   S711A_WELD_BUFF_DATA1.RBT13_BT_CODE_NO := W#16#0;
   S711A_WELD_BUFF_DATA1.RBT13_WELD_COUNT := W#16#0;
   S711A_WELD_BUFF_DATA1.RBT14_BT_CODE_NO := W#16#0;
   S711A_WELD_BUFF_DATA1.RBT14_WELD_COUNT := W#16#0;
   S711A_WELD_BUFF_DATA1.RBT15_BT_CODE_NO := W#16#0;
   S711A_WELD_BUFF_DATA1.RBT15_WELD_COUNT := W#16#0;
   S711A_WELD_BUFF_DATA1.RBT16_BT_CODE_NO := W#16#0;
   S711A_WELD_BUFF_DATA1.RBT16_WELD_COUNT := W#16#0;
   S711A_WELD_BUFF_DATA1.RBT17_BT_CODE_NO := W#16#0;
   S711A_WELD_BUFF_DATA1.RBT17_WELD_COUNT := W#16#0;
   S711A_WELD_BUFF_DATA1.RBT18_BT_CODE_NO := W#16#0;
   S711A_WELD_BUFF_DATA1.RBT18_WELD_COUNT := W#16#0;
   S711A_WELD_BUFF_DATA1.RBT19_BT_CODE_NO := W#16#0;
   S711A_WELD_BUFF_DATA1.RBT19_WELD_COUNT := W#16#0;
   S711A_WELD_BUFF_DATA1.RBT20_BT_CODE_NO := W#16#0;
   S711A_WELD_BUFF_DATA1.RBT20_WELD_COUNT := W#16#0;
   S711A_WELD_BUFF_DATA1.RBT21_BT_CODE_NO := W#16#0;
   S711A_WELD_BUFF_DATA1.RBT21_WELD_COUNT := W#16#0;
   S711A_WELD_BUFF_DATA1.RBT22_BT_CODE_NO := W#16#0;
   S711A_WELD_BUFF_DATA1.RBT22_WELD_COUNT := W#16#0;
   S711A_WELD_BUFF_DATA1.RBT23_BT_CODE_NO := W#16#0;
   S711A_WELD_BUFF_DATA1.RBT23_WELD_COUNT := W#16#0;
   S711A_WELD_BUFF_DATA1.RBT24_BT_CODE_NO := W#16#0;
   S711A_WELD_BUFF_DATA1.RBT24_WELD_COUNT := W#16#0;
   S711A_WELD_BUFF_DATA1.WELD_DETERMINES_RESULT := W#16#0;
   S711A_WELD_BUFF_DATA1.WELD_CHECK_SUM := W#16#0;
   S711A_WELD_BUFF_DATA1.SPARE1 := W#16#0;
   S711A_WELD_BUFF_DATA2.STATION_MAIN := W#16#0;
   S711A_WELD_BUFF_DATA2.DISTINCTION_LH_RH := W#16#0;
   S711A_WELD_BUFF_DATA2.STAION_NUMBER := W#16#0;
   S711A_WELD_BUFF_DATA2.VIN_NUMBER1 := W#16#0;
   S711A_WELD_BUFF_DATA2.VIN_NUMBER2 := W#16#0;
   S711A_WELD_BUFF_DATA2.VIN_NUMBER3 := W#16#0;
   S711A_WELD_BUFF_DATA2.VIN_NUMBER4 := W#16#0;
   S711A_WELD_BUFF_DATA2.SEQ_NUMBER1 := W#16#0;
   S711A_WELD_BUFF_DATA2.SEQ_NUMBER2 := W#16#0;
   S711A_WELD_BUFF_DATA2.RBT1_BT_CODE_NO := W#16#0;
   S711A_WELD_BUFF_DATA2.RBT1_WELD_COUNT := W#16#0;
   S711A_WELD_BUFF_DATA2.RBT2_BT_CODE_NO := W#16#0;
   S711A_WELD_BUFF_DATA2.RBT2_WELD_COUNT := W#16#0;
   S711A_WELD_BUFF_DATA2.RBT3_BT_CODE_NO := W#16#0;
   S711A_WELD_BUFF_DATA2.RBT3_WELD_COUNT := W#16#0;
   S711A_WELD_BUFF_DATA2.RBT4_BT_CODE_NO := W#16#0;
   S711A_WELD_BUFF_DATA2.RBT4_WELD_COUNT := W#16#0;
   S711A_WELD_BUFF_DATA2.RBT5_BT_CODE_NO := W#16#0;
   S711A_WELD_BUFF_DATA2.RBT5_WELD_COUNT := W#16#0;
   S711A_WELD_BUFF_DATA2.RBT6_BT_CODE_NO := W#16#0;
   S711A_WELD_BUFF_DATA2.RBT6_WELD_COUNT := W#16#0;
   S711A_WELD_BUFF_DATA2.RBT7_BT_CODE_NO := W#16#0;
   S711A_WELD_BUFF_DATA2.RBT7_WELD_COUNT := W#16#0;
   S711A_WELD_BUFF_DATA2.RBT8_BT_CODE_NO := W#16#0;
   S711A_WELD_BUFF_DATA2.RBT8_WELD_COUNT := W#16#0;
   S711A_WELD_BUFF_DATA2.RBT9_BT_CODE_NO := W#16#0;
   S711A_WELD_BUFF_DATA2.RBT9_WELD_COUNT := W#16#0;
   S711A_WELD_BUFF_DATA2.RBT10_BT_CODE_NO := W#16#0;
   S711A_WELD_BUFF_DATA2.RBT10_WELD_COUNT := W#16#0;
   S711A_WELD_BUFF_DATA2.RBT11_BT_CODE_NO := W#16#0;
   S711A_WELD_BUFF_DATA2.RBT11_WELD_COUNT := W#16#0;
   S711A_WELD_BUFF_DATA2.RBT12_BT_CODE_NO := W#16#0;
   S711A_WELD_BUFF_DATA2.RBT12_WELD_COUNT := W#16#0;
   S711A_WELD_BUFF_DATA2.RBT13_BT_CODE_NO := W#16#0;
   S711A_WELD_BUFF_DATA2.RBT13_WELD_COUNT := W#16#0;
   S711A_WELD_BUFF_DATA2.RBT14_BT_CODE_NO := W#16#0;
   S711A_WELD_BUFF_DATA2.RBT14_WELD_COUNT := W#16#0;
   S711A_WELD_BUFF_DATA2.RBT15_BT_CODE_NO := W#16#0;
   S711A_WELD_BUFF_DATA2.RBT15_WELD_COUNT := W#16#0;
   S711A_WELD_BUFF_DATA2.RBT16_BT_CODE_NO := W#16#0;
   S711A_WELD_BUFF_DATA2.RBT16_WELD_COUNT := W#16#0;
   S711A_WELD_BUFF_DATA2.RBT17_BT_CODE_NO := W#16#0;
   S711A_WELD_BUFF_DATA2.RBT17_WELD_COUNT := W#16#0;
   S711A_WELD_BUFF_DATA2.RBT18_BT_CODE_NO := W#16#0;
   S711A_WELD_BUFF_DATA2.RBT18_WELD_COUNT := W#16#0;
   S711A_WELD_BUFF_DATA2.RBT19_BT_CODE_NO := W#16#0;
   S711A_WELD_BUFF_DATA2.RBT19_WELD_COUNT := W#16#0;
   S711A_WELD_BUFF_DATA2.RBT20_BT_CODE_NO := W#16#0;
   S711A_WELD_BUFF_DATA2.RBT20_WELD_COUNT := W#16#0;
   S711A_WELD_BUFF_DATA2.RBT21_BT_CODE_NO := W#16#0;
   S711A_WELD_BUFF_DATA2.RBT21_WELD_COUNT := W#16#0;
   S711A_WELD_BUFF_DATA2.RBT22_BT_CODE_NO := W#16#0;
   S711A_WELD_BUFF_DATA2.RBT22_WELD_COUNT := W#16#0;
   S711A_WELD_BUFF_DATA2.RBT23_BT_CODE_NO := W#16#0;
   S711A_WELD_BUFF_DATA2.RBT23_WELD_COUNT := W#16#0;
   S711A_WELD_BUFF_DATA2.RBT24_BT_CODE_NO := W#16#0;
   S711A_WELD_BUFF_DATA2.RBT24_WELD_COUNT := W#16#0;
   S711A_WELD_BUFF_DATA2.WELD_DETERMINES_RESULT := W#16#0;
   S711A_WELD_BUFF_DATA2.WELD_CHECK_SUM := W#16#0;
   S711A_WELD_BUFF_DATA2.SPARE1 := W#16#0;
   S711A_WELD_BUFF_DATA3.STATION_MAIN := W#16#0;
   S711A_WELD_BUFF_DATA3.DISTINCTION_LH_RH := W#16#0;
   S711A_WELD_BUFF_DATA3.STAION_NUMBER := W#16#0;
   S711A_WELD_BUFF_DATA3.VIN_NUMBER1 := W#16#0;
   S711A_WELD_BUFF_DATA3.VIN_NUMBER2 := W#16#0;
   S711A_WELD_BUFF_DATA3.VIN_NUMBER3 := W#16#0;
   S711A_WELD_BUFF_DATA3.VIN_NUMBER4 := W#16#0;
   S711A_WELD_BUFF_DATA3.SEQ_NUMBER1 := W#16#0;
   S711A_WELD_BUFF_DATA3.SEQ_NUMBER2 := W#16#0;
   S711A_WELD_BUFF_DATA3.RBT1_BT_CODE_NO := W#16#0;
   S711A_WELD_BUFF_DATA3.RBT1_WELD_COUNT := W#16#0;
   S711A_WELD_BUFF_DATA3.RBT2_BT_CODE_NO := W#16#0;
   S711A_WELD_BUFF_DATA3.RBT2_WELD_COUNT := W#16#0;
   S711A_WELD_BUFF_DATA3.RBT3_BT_CODE_NO := W#16#0;
   S711A_WELD_BUFF_DATA3.RBT3_WELD_COUNT := W#16#0;
   S711A_WELD_BUFF_DATA3.RBT4_BT_CODE_NO := W#16#0;
   S711A_WELD_BUFF_DATA3.RBT4_WELD_COUNT := W#16#0;
   S711A_WELD_BUFF_DATA3.RBT5_BT_CODE_NO := W#16#0;
   S711A_WELD_BUFF_DATA3.RBT5_WELD_COUNT := W#16#0;
   S711A_WELD_BUFF_DATA3.RBT6_BT_CODE_NO := W#16#0;
   S711A_WELD_BUFF_DATA3.RBT6_WELD_COUNT := W#16#0;
   S711A_WELD_BUFF_DATA3.RBT7_BT_CODE_NO := W#16#0;
   S711A_WELD_BUFF_DATA3.RBT7_WELD_COUNT := W#16#0;
   S711A_WELD_BUFF_DATA3.RBT8_BT_CODE_NO := W#16#0;
   S711A_WELD_BUFF_DATA3.RBT8_WELD_COUNT := W#16#0;
   S711A_WELD_BUFF_DATA3.RBT9_BT_CODE_NO := W#16#0;
   S711A_WELD_BUFF_DATA3.RBT9_WELD_COUNT := W#16#0;
   S711A_WELD_BUFF_DATA3.RBT10_BT_CODE_NO := W#16#0;
   S711A_WELD_BUFF_DATA3.RBT10_WELD_COUNT := W#16#0;
   S711A_WELD_BUFF_DATA3.RBT11_BT_CODE_NO := W#16#0;
   S711A_WELD_BUFF_DATA3.RBT11_WELD_COUNT := W#16#0;
   S711A_WELD_BUFF_DATA3.RBT12_BT_CODE_NO := W#16#0;
   S711A_WELD_BUFF_DATA3.RBT12_WELD_COUNT := W#16#0;
   S711A_WELD_BUFF_DATA3.RBT13_BT_CODE_NO := W#16#0;
   S711A_WELD_BUFF_DATA3.RBT13_WELD_COUNT := W#16#0;
   S711A_WELD_BUFF_DATA3.RBT14_BT_CODE_NO := W#16#0;
   S711A_WELD_BUFF_DATA3.RBT14_WELD_COUNT := W#16#0;
   S711A_WELD_BUFF_DATA3.RBT15_BT_CODE_NO := W#16#0;
   S711A_WELD_BUFF_DATA3.RBT15_WELD_COUNT := W#16#0;
   S711A_WELD_BUFF_DATA3.RBT16_BT_CODE_NO := W#16#0;
   S711A_WELD_BUFF_DATA3.RBT16_WELD_COUNT := W#16#0;
   S711A_WELD_BUFF_DATA3.RBT17_BT_CODE_NO := W#16#0;
   S711A_WELD_BUFF_DATA3.RBT17_WELD_COUNT := W#16#0;
   S711A_WELD_BUFF_DATA3.RBT18_BT_CODE_NO := W#16#0;
   S711A_WELD_BUFF_DATA3.RBT18_WELD_COUNT := W#16#0;
   S711A_WELD_BUFF_DATA3.RBT19_BT_CODE_NO := W#16#0;
   S711A_WELD_BUFF_DATA3.RBT19_WELD_COUNT := W#16#0;
   S711A_WELD_BUFF_DATA3.RBT20_BT_CODE_NO := W#16#0;
   S711A_WELD_BUFF_DATA3.RBT20_WELD_COUNT := W#16#0;
   S711A_WELD_BUFF_DATA3.RBT21_BT_CODE_NO := W#16#0;
   S711A_WELD_BUFF_DATA3.RBT21_WELD_COUNT := W#16#0;
   S711A_WELD_BUFF_DATA3.RBT22_BT_CODE_NO := W#16#0;
   S711A_WELD_BUFF_DATA3.RBT22_WELD_COUNT := W#16#0;
   S711A_WELD_BUFF_DATA3.RBT23_BT_CODE_NO := W#16#0;
   S711A_WELD_BUFF_DATA3.RBT23_WELD_COUNT := W#16#0;
   S711A_WELD_BUFF_DATA3.RBT24_BT_CODE_NO := W#16#0;
   S711A_WELD_BUFF_DATA3.RBT24_WELD_COUNT := W#16#0;
   S711A_WELD_BUFF_DATA3.WELD_DETERMINES_RESULT := W#16#0;
   S711A_WELD_BUFF_DATA3.WELD_CHECK_SUM := W#16#0;
   S711A_WELD_BUFF_DATA3.SPARE1 := W#16#0;
   S711A_WELD_BUFF_DATA4.STATION_MAIN := W#16#0;
   S711A_WELD_BUFF_DATA4.DISTINCTION_LH_RH := W#16#0;
   S711A_WELD_BUFF_DATA4.STAION_NUMBER := W#16#0;
   S711A_WELD_BUFF_DATA4.VIN_NUMBER1 := W#16#0;
   S711A_WELD_BUFF_DATA4.VIN_NUMBER2 := W#16#0;
   S711A_WELD_BUFF_DATA4.VIN_NUMBER3 := W#16#0;
   S711A_WELD_BUFF_DATA4.VIN_NUMBER4 := W#16#0;
   S711A_WELD_BUFF_DATA4.SEQ_NUMBER1 := W#16#0;
   S711A_WELD_BUFF_DATA4.SEQ_NUMBER2 := W#16#0;
   S711A_WELD_BUFF_DATA4.RBT1_BT_CODE_NO := W#16#0;
   S711A_WELD_BUFF_DATA4.RBT1_WELD_COUNT := W#16#0;
   S711A_WELD_BUFF_DATA4.RBT2_BT_CODE_NO := W#16#0;
   S711A_WELD_BUFF_DATA4.RBT2_WELD_COUNT := W#16#0;
   S711A_WELD_BUFF_DATA4.RBT3_BT_CODE_NO := W#16#0;
   S711A_WELD_BUFF_DATA4.RBT3_WELD_COUNT := W#16#0;
   S711A_WELD_BUFF_DATA4.RBT4_BT_CODE_NO := W#16#0;
   S711A_WELD_BUFF_DATA4.RBT4_WELD_COUNT := W#16#0;
   S711A_WELD_BUFF_DATA4.RBT5_BT_CODE_NO := W#16#0;
   S711A_WELD_BUFF_DATA4.RBT5_WELD_COUNT := W#16#0;
   S711A_WELD_BUFF_DATA4.RBT6_BT_CODE_NO := W#16#0;
   S711A_WELD_BUFF_DATA4.RBT6_WELD_COUNT := W#16#0;
   S711A_WELD_BUFF_DATA4.RBT7_BT_CODE_NO := W#16#0;
   S711A_WELD_BUFF_DATA4.RBT7_WELD_COUNT := W#16#0;
   S711A_WELD_BUFF_DATA4.RBT8_BT_CODE_NO := W#16#0;
   S711A_WELD_BUFF_DATA4.RBT8_WELD_COUNT := W#16#0;
   S711A_WELD_BUFF_DATA4.RBT9_BT_CODE_NO := W#16#0;
   S711A_WELD_BUFF_DATA4.RBT9_WELD_COUNT := W#16#0;
   S711A_WELD_BUFF_DATA4.RBT10_BT_CODE_NO := W#16#0;
   S711A_WELD_BUFF_DATA4.RBT10_WELD_COUNT := W#16#0;
   S711A_WELD_BUFF_DATA4.RBT11_BT_CODE_NO := W#16#0;
   S711A_WELD_BUFF_DATA4.RBT11_WELD_COUNT := W#16#0;
   S711A_WELD_BUFF_DATA4.RBT12_BT_CODE_NO := W#16#0;
   S711A_WELD_BUFF_DATA4.RBT12_WELD_COUNT := W#16#0;
   S711A_WELD_BUFF_DATA4.RBT13_BT_CODE_NO := W#16#0;
   S711A_WELD_BUFF_DATA4.RBT13_WELD_COUNT := W#16#0;
   S711A_WELD_BUFF_DATA4.RBT14_BT_CODE_NO := W#16#0;
   S711A_WELD_BUFF_DATA4.RBT14_WELD_COUNT := W#16#0;
   S711A_WELD_BUFF_DATA4.RBT15_BT_CODE_NO := W#16#0;
   S711A_WELD_BUFF_DATA4.RBT15_WELD_COUNT := W#16#0;
   S711A_WELD_BUFF_DATA4.RBT16_BT_CODE_NO := W#16#0;
   S711A_WELD_BUFF_DATA4.RBT16_WELD_COUNT := W#16#0;
   S711A_WELD_BUFF_DATA4.RBT17_BT_CODE_NO := W#16#0;
   S711A_WELD_BUFF_DATA4.RBT17_WELD_COUNT := W#16#0;
   S711A_WELD_BUFF_DATA4.RBT18_BT_CODE_NO := W#16#0;
   S711A_WELD_BUFF_DATA4.RBT18_WELD_COUNT := W#16#0;
   S711A_WELD_BUFF_DATA4.RBT19_BT_CODE_NO := W#16#0;
   S711A_WELD_BUFF_DATA4.RBT19_WELD_COUNT := W#16#0;
   S711A_WELD_BUFF_DATA4.RBT20_BT_CODE_NO := W#16#0;
   S711A_WELD_BUFF_DATA4.RBT20_WELD_COUNT := W#16#0;
   S711A_WELD_BUFF_DATA4.RBT21_BT_CODE_NO := W#16#0;
   S711A_WELD_BUFF_DATA4.RBT21_WELD_COUNT := W#16#0;
   S711A_WELD_BUFF_DATA4.RBT22_BT_CODE_NO := W#16#0;
   S711A_WELD_BUFF_DATA4.RBT22_WELD_COUNT := W#16#0;
   S711A_WELD_BUFF_DATA4.RBT23_BT_CODE_NO := W#16#0;
   S711A_WELD_BUFF_DATA4.RBT23_WELD_COUNT := W#16#0;
   S711A_WELD_BUFF_DATA4.RBT24_BT_CODE_NO := W#16#0;
   S711A_WELD_BUFF_DATA4.RBT24_WELD_COUNT := W#16#0;
   S711A_WELD_BUFF_DATA4.WELD_DETERMINES_RESULT := W#16#0;
   S711A_WELD_BUFF_DATA4.WELD_CHECK_SUM := W#16#0;
   S711A_WELD_BUFF_DATA4.SPARE1 := W#16#0;
   S711A_WELD_BUFF_DATA5.STATION_MAIN := W#16#0;
   S711A_WELD_BUFF_DATA5.DISTINCTION_LH_RH := W#16#0;
   S711A_WELD_BUFF_DATA5.STAION_NUMBER := W#16#0;
   S711A_WELD_BUFF_DATA5.VIN_NUMBER1 := W#16#0;
   S711A_WELD_BUFF_DATA5.VIN_NUMBER2 := W#16#0;
   S711A_WELD_BUFF_DATA5.VIN_NUMBER3 := W#16#0;
   S711A_WELD_BUFF_DATA5.VIN_NUMBER4 := W#16#0;
   S711A_WELD_BUFF_DATA5.SEQ_NUMBER1 := W#16#0;
   S711A_WELD_BUFF_DATA5.SEQ_NUMBER2 := W#16#0;
   S711A_WELD_BUFF_DATA5.RBT1_BT_CODE_NO := W#16#0;
   S711A_WELD_BUFF_DATA5.RBT1_WELD_COUNT := W#16#0;
   S711A_WELD_BUFF_DATA5.RBT2_BT_CODE_NO := W#16#0;
   S711A_WELD_BUFF_DATA5.RBT2_WELD_COUNT := W#16#0;
   S711A_WELD_BUFF_DATA5.RBT3_BT_CODE_NO := W#16#0;
   S711A_WELD_BUFF_DATA5.RBT3_WELD_COUNT := W#16#0;
   S711A_WELD_BUFF_DATA5.RBT4_BT_CODE_NO := W#16#0;
   S711A_WELD_BUFF_DATA5.RBT4_WELD_COUNT := W#16#0;
   S711A_WELD_BUFF_DATA5.RBT5_BT_CODE_NO := W#16#0;
   S711A_WELD_BUFF_DATA5.RBT5_WELD_COUNT := W#16#0;
   S711A_WELD_BUFF_DATA5.RBT6_BT_CODE_NO := W#16#0;
   S711A_WELD_BUFF_DATA5.RBT6_WELD_COUNT := W#16#0;
   S711A_WELD_BUFF_DATA5.RBT7_BT_CODE_NO := W#16#0;
   S711A_WELD_BUFF_DATA5.RBT7_WELD_COUNT := W#16#0;
   S711A_WELD_BUFF_DATA5.RBT8_BT_CODE_NO := W#16#0;
   S711A_WELD_BUFF_DATA5.RBT8_WELD_COUNT := W#16#0;
   S711A_WELD_BUFF_DATA5.RBT9_BT_CODE_NO := W#16#0;
   S711A_WELD_BUFF_DATA5.RBT9_WELD_COUNT := W#16#0;
   S711A_WELD_BUFF_DATA5.RBT10_BT_CODE_NO := W#16#0;
   S711A_WELD_BUFF_DATA5.RBT10_WELD_COUNT := W#16#0;
   S711A_WELD_BUFF_DATA5.RBT11_BT_CODE_NO := W#16#0;
   S711A_WELD_BUFF_DATA5.RBT11_WELD_COUNT := W#16#0;
   S711A_WELD_BUFF_DATA5.RBT12_BT_CODE_NO := W#16#0;
   S711A_WELD_BUFF_DATA5.RBT12_WELD_COUNT := W#16#0;
   S711A_WELD_BUFF_DATA5.RBT13_BT_CODE_NO := W#16#0;
   S711A_WELD_BUFF_DATA5.RBT13_WELD_COUNT := W#16#0;
   S711A_WELD_BUFF_DATA5.RBT14_BT_CODE_NO := W#16#0;
   S711A_WELD_BUFF_DATA5.RBT14_WELD_COUNT := W#16#0;
   S711A_WELD_BUFF_DATA5.RBT15_BT_CODE_NO := W#16#0;
   S711A_WELD_BUFF_DATA5.RBT15_WELD_COUNT := W#16#0;
   S711A_WELD_BUFF_DATA5.RBT16_BT_CODE_NO := W#16#0;
   S711A_WELD_BUFF_DATA5.RBT16_WELD_COUNT := W#16#0;
   S711A_WELD_BUFF_DATA5.RBT17_BT_CODE_NO := W#16#0;
   S711A_WELD_BUFF_DATA5.RBT17_WELD_COUNT := W#16#0;
   S711A_WELD_BUFF_DATA5.RBT18_BT_CODE_NO := W#16#0;
   S711A_WELD_BUFF_DATA5.RBT18_WELD_COUNT := W#16#0;
   S711A_WELD_BUFF_DATA5.RBT19_BT_CODE_NO := W#16#0;
   S711A_WELD_BUFF_DATA5.RBT19_WELD_COUNT := W#16#0;
   S711A_WELD_BUFF_DATA5.RBT20_BT_CODE_NO := W#16#0;
   S711A_WELD_BUFF_DATA5.RBT20_WELD_COUNT := W#16#0;
   S711A_WELD_BUFF_DATA5.RBT21_BT_CODE_NO := W#16#0;
   S711A_WELD_BUFF_DATA5.RBT21_WELD_COUNT := W#16#0;
   S711A_WELD_BUFF_DATA5.RBT22_BT_CODE_NO := W#16#0;
   S711A_WELD_BUFF_DATA5.RBT22_WELD_COUNT := W#16#0;
   S711A_WELD_BUFF_DATA5.RBT23_BT_CODE_NO := W#16#0;
   S711A_WELD_BUFF_DATA5.RBT23_WELD_COUNT := W#16#0;
   S711A_WELD_BUFF_DATA5.RBT24_BT_CODE_NO := W#16#0;
   S711A_WELD_BUFF_DATA5.RBT24_WELD_COUNT := W#16#0;
   S711A_WELD_BUFF_DATA5.WELD_DETERMINES_RESULT := W#16#0;
   S711A_WELD_BUFF_DATA5.WELD_CHECK_SUM := W#16#0;
   S711A_WELD_BUFF_DATA5.SPARE1 := W#16#0;
   S711A_WELD_BUFF_DATA6.STATION_MAIN := W#16#0;
   S711A_WELD_BUFF_DATA6.DISTINCTION_LH_RH := W#16#0;
   S711A_WELD_BUFF_DATA6.STAION_NUMBER := W#16#0;
   S711A_WELD_BUFF_DATA6.VIN_NUMBER1 := W#16#0;
   S711A_WELD_BUFF_DATA6.VIN_NUMBER2 := W#16#0;
   S711A_WELD_BUFF_DATA6.VIN_NUMBER3 := W#16#0;
   S711A_WELD_BUFF_DATA6.VIN_NUMBER4 := W#16#0;
   S711A_WELD_BUFF_DATA6.SEQ_NUMBER1 := W#16#0;
   S711A_WELD_BUFF_DATA6.SEQ_NUMBER2 := W#16#0;
   S711A_WELD_BUFF_DATA6.RBT1_BT_CODE_NO := W#16#0;
   S711A_WELD_BUFF_DATA6.RBT1_WELD_COUNT := W#16#0;
   S711A_WELD_BUFF_DATA6.RBT2_BT_CODE_NO := W#16#0;
   S711A_WELD_BUFF_DATA6.RBT2_WELD_COUNT := W#16#0;
   S711A_WELD_BUFF_DATA6.RBT3_BT_CODE_NO := W#16#0;
   S711A_WELD_BUFF_DATA6.RBT3_WELD_COUNT := W#16#0;
   S711A_WELD_BUFF_DATA6.RBT4_BT_CODE_NO := W#16#0;
   S711A_WELD_BUFF_DATA6.RBT4_WELD_COUNT := W#16#0;
   S711A_WELD_BUFF_DATA6.RBT5_BT_CODE_NO := W#16#0;
   S711A_WELD_BUFF_DATA6.RBT5_WELD_COUNT := W#16#0;
   S711A_WELD_BUFF_DATA6.RBT6_BT_CODE_NO := W#16#0;
   S711A_WELD_BUFF_DATA6.RBT6_WELD_COUNT := W#16#0;
   S711A_WELD_BUFF_DATA6.RBT7_BT_CODE_NO := W#16#0;
   S711A_WELD_BUFF_DATA6.RBT7_WELD_COUNT := W#16#0;
   S711A_WELD_BUFF_DATA6.RBT8_BT_CODE_NO := W#16#0;
   S711A_WELD_BUFF_DATA6.RBT8_WELD_COUNT := W#16#0;
   S711A_WELD_BUFF_DATA6.RBT9_BT_CODE_NO := W#16#0;
   S711A_WELD_BUFF_DATA6.RBT9_WELD_COUNT := W#16#0;
   S711A_WELD_BUFF_DATA6.RBT10_BT_CODE_NO := W#16#0;
   S711A_WELD_BUFF_DATA6.RBT10_WELD_COUNT := W#16#0;
   S711A_WELD_BUFF_DATA6.RBT11_BT_CODE_NO := W#16#0;
   S711A_WELD_BUFF_DATA6.RBT11_WELD_COUNT := W#16#0;
   S711A_WELD_BUFF_DATA6.RBT12_BT_CODE_NO := W#16#0;
   S711A_WELD_BUFF_DATA6.RBT12_WELD_COUNT := W#16#0;
   S711A_WELD_BUFF_DATA6.RBT13_BT_CODE_NO := W#16#0;
   S711A_WELD_BUFF_DATA6.RBT13_WELD_COUNT := W#16#0;
   S711A_WELD_BUFF_DATA6.RBT14_BT_CODE_NO := W#16#0;
   S711A_WELD_BUFF_DATA6.RBT14_WELD_COUNT := W#16#0;
   S711A_WELD_BUFF_DATA6.RBT15_BT_CODE_NO := W#16#0;
   S711A_WELD_BUFF_DATA6.RBT15_WELD_COUNT := W#16#0;
   S711A_WELD_BUFF_DATA6.RBT16_BT_CODE_NO := W#16#0;
   S711A_WELD_BUFF_DATA6.RBT16_WELD_COUNT := W#16#0;
   S711A_WELD_BUFF_DATA6.RBT17_BT_CODE_NO := W#16#0;
   S711A_WELD_BUFF_DATA6.RBT17_WELD_COUNT := W#16#0;
   S711A_WELD_BUFF_DATA6.RBT18_BT_CODE_NO := W#16#0;
   S711A_WELD_BUFF_DATA6.RBT18_WELD_COUNT := W#16#0;
   S711A_WELD_BUFF_DATA6.RBT19_BT_CODE_NO := W#16#0;
   S711A_WELD_BUFF_DATA6.RBT19_WELD_COUNT := W#16#0;
   S711A_WELD_BUFF_DATA6.RBT20_BT_CODE_NO := W#16#0;
   S711A_WELD_BUFF_DATA6.RBT20_WELD_COUNT := W#16#0;
   S711A_WELD_BUFF_DATA6.RBT21_BT_CODE_NO := W#16#0;
   S711A_WELD_BUFF_DATA6.RBT21_WELD_COUNT := W#16#0;
   S711A_WELD_BUFF_DATA6.RBT22_BT_CODE_NO := W#16#0;
   S711A_WELD_BUFF_DATA6.RBT22_WELD_COUNT := W#16#0;
   S711A_WELD_BUFF_DATA6.RBT23_BT_CODE_NO := W#16#0;
   S711A_WELD_BUFF_DATA6.RBT23_WELD_COUNT := W#16#0;
   S711A_WELD_BUFF_DATA6.RBT24_BT_CODE_NO := W#16#0;
   S711A_WELD_BUFF_DATA6.RBT24_WELD_COUNT := W#16#0;
   S711A_WELD_BUFF_DATA6.WELD_DETERMINES_RESULT := W#16#0;
   S711A_WELD_BUFF_DATA6.WELD_CHECK_SUM := W#16#0;
   S711A_WELD_BUFF_DATA6.SPARE1 := W#16#0;
   S711A_WELD_BUFF_DATA7.STATION_MAIN := W#16#0;
   S711A_WELD_BUFF_DATA7.DISTINCTION_LH_RH := W#16#0;
   S711A_WELD_BUFF_DATA7.STAION_NUMBER := W#16#0;
   S711A_WELD_BUFF_DATA7.VIN_NUMBER1 := W#16#0;
   S711A_WELD_BUFF_DATA7.VIN_NUMBER2 := W#16#0;
   S711A_WELD_BUFF_DATA7.VIN_NUMBER3 := W#16#0;
   S711A_WELD_BUFF_DATA7.VIN_NUMBER4 := W#16#0;
   S711A_WELD_BUFF_DATA7.SEQ_NUMBER1 := W#16#0;
   S711A_WELD_BUFF_DATA7.SEQ_NUMBER2 := W#16#0;
   S711A_WELD_BUFF_DATA7.RBT1_BT_CODE_NO := W#16#0;
   S711A_WELD_BUFF_DATA7.RBT1_WELD_COUNT := W#16#0;
   S711A_WELD_BUFF_DATA7.RBT2_BT_CODE_NO := W#16#0;
   S711A_WELD_BUFF_DATA7.RBT2_WELD_COUNT := W#16#0;
   S711A_WELD_BUFF_DATA7.RBT3_BT_CODE_NO := W#16#0;
   S711A_WELD_BUFF_DATA7.RBT3_WELD_COUNT := W#16#0;
   S711A_WELD_BUFF_DATA7.RBT4_BT_CODE_NO := W#16#0;
   S711A_WELD_BUFF_DATA7.RBT4_WELD_COUNT := W#16#0;
   S711A_WELD_BUFF_DATA7.RBT5_BT_CODE_NO := W#16#0;
   S711A_WELD_BUFF_DATA7.RBT5_WELD_COUNT := W#16#0;
   S711A_WELD_BUFF_DATA7.RBT6_BT_CODE_NO := W#16#0;
   S711A_WELD_BUFF_DATA7.RBT6_WELD_COUNT := W#16#0;
   S711A_WELD_BUFF_DATA7.RBT7_BT_CODE_NO := W#16#0;
   S711A_WELD_BUFF_DATA7.RBT7_WELD_COUNT := W#16#0;
   S711A_WELD_BUFF_DATA7.RBT8_BT_CODE_NO := W#16#0;
   S711A_WELD_BUFF_DATA7.RBT8_WELD_COUNT := W#16#0;
   S711A_WELD_BUFF_DATA7.RBT9_BT_CODE_NO := W#16#0;
   S711A_WELD_BUFF_DATA7.RBT9_WELD_COUNT := W#16#0;
   S711A_WELD_BUFF_DATA7.RBT10_BT_CODE_NO := W#16#0;
   S711A_WELD_BUFF_DATA7.RBT10_WELD_COUNT := W#16#0;
   S711A_WELD_BUFF_DATA7.RBT11_BT_CODE_NO := W#16#0;
   S711A_WELD_BUFF_DATA7.RBT11_WELD_COUNT := W#16#0;
   S711A_WELD_BUFF_DATA7.RBT12_BT_CODE_NO := W#16#0;
   S711A_WELD_BUFF_DATA7.RBT12_WELD_COUNT := W#16#0;
   S711A_WELD_BUFF_DATA7.RBT13_BT_CODE_NO := W#16#0;
   S711A_WELD_BUFF_DATA7.RBT13_WELD_COUNT := W#16#0;
   S711A_WELD_BUFF_DATA7.RBT14_BT_CODE_NO := W#16#0;
   S711A_WELD_BUFF_DATA7.RBT14_WELD_COUNT := W#16#0;
   S711A_WELD_BUFF_DATA7.RBT15_BT_CODE_NO := W#16#0;
   S711A_WELD_BUFF_DATA7.RBT15_WELD_COUNT := W#16#0;
   S711A_WELD_BUFF_DATA7.RBT16_BT_CODE_NO := W#16#0;
   S711A_WELD_BUFF_DATA7.RBT16_WELD_COUNT := W#16#0;
   S711A_WELD_BUFF_DATA7.RBT17_BT_CODE_NO := W#16#0;
   S711A_WELD_BUFF_DATA7.RBT17_WELD_COUNT := W#16#0;
   S711A_WELD_BUFF_DATA7.RBT18_BT_CODE_NO := W#16#0;
   S711A_WELD_BUFF_DATA7.RBT18_WELD_COUNT := W#16#0;
   S711A_WELD_BUFF_DATA7.RBT19_BT_CODE_NO := W#16#0;
   S711A_WELD_BUFF_DATA7.RBT19_WELD_COUNT := W#16#0;
   S711A_WELD_BUFF_DATA7.RBT20_BT_CODE_NO := W#16#0;
   S711A_WELD_BUFF_DATA7.RBT20_WELD_COUNT := W#16#0;
   S711A_WELD_BUFF_DATA7.RBT21_BT_CODE_NO := W#16#0;
   S711A_WELD_BUFF_DATA7.RBT21_WELD_COUNT := W#16#0;
   S711A_WELD_BUFF_DATA7.RBT22_BT_CODE_NO := W#16#0;
   S711A_WELD_BUFF_DATA7.RBT22_WELD_COUNT := W#16#0;
   S711A_WELD_BUFF_DATA7.RBT23_BT_CODE_NO := W#16#0;
   S711A_WELD_BUFF_DATA7.RBT23_WELD_COUNT := W#16#0;
   S711A_WELD_BUFF_DATA7.RBT24_BT_CODE_NO := W#16#0;
   S711A_WELD_BUFF_DATA7.RBT24_WELD_COUNT := W#16#0;
   S711A_WELD_BUFF_DATA7.WELD_DETERMINES_RESULT := W#16#0;
   S711A_WELD_BUFF_DATA7.WELD_CHECK_SUM := W#16#0;
   S711A_WELD_BUFF_DATA7.SPARE1 := W#16#0;
   S711A_WELD_BUFF_DATA8.STATION_MAIN := W#16#0;
   S711A_WELD_BUFF_DATA8.DISTINCTION_LH_RH := W#16#0;
   S711A_WELD_BUFF_DATA8.STAION_NUMBER := W#16#0;
   S711A_WELD_BUFF_DATA8.VIN_NUMBER1 := W#16#0;
   S711A_WELD_BUFF_DATA8.VIN_NUMBER2 := W#16#0;
   S711A_WELD_BUFF_DATA8.VIN_NUMBER3 := W#16#0;
   S711A_WELD_BUFF_DATA8.VIN_NUMBER4 := W#16#0;
   S711A_WELD_BUFF_DATA8.SEQ_NUMBER1 := W#16#0;
   S711A_WELD_BUFF_DATA8.SEQ_NUMBER2 := W#16#0;
   S711A_WELD_BUFF_DATA8.RBT1_BT_CODE_NO := W#16#0;
   S711A_WELD_BUFF_DATA8.RBT1_WELD_COUNT := W#16#0;
   S711A_WELD_BUFF_DATA8.RBT2_BT_CODE_NO := W#16#0;
   S711A_WELD_BUFF_DATA8.RBT2_WELD_COUNT := W#16#0;
   S711A_WELD_BUFF_DATA8.RBT3_BT_CODE_NO := W#16#0;
   S711A_WELD_BUFF_DATA8.RBT3_WELD_COUNT := W#16#0;
   S711A_WELD_BUFF_DATA8.RBT4_BT_CODE_NO := W#16#0;
   S711A_WELD_BUFF_DATA8.RBT4_WELD_COUNT := W#16#0;
   S711A_WELD_BUFF_DATA8.RBT5_BT_CODE_NO := W#16#0;
   S711A_WELD_BUFF_DATA8.RBT5_WELD_COUNT := W#16#0;
   S711A_WELD_BUFF_DATA8.RBT6_BT_CODE_NO := W#16#0;
   S711A_WELD_BUFF_DATA8.RBT6_WELD_COUNT := W#16#0;
   S711A_WELD_BUFF_DATA8.RBT7_BT_CODE_NO := W#16#0;
   S711A_WELD_BUFF_DATA8.RBT7_WELD_COUNT := W#16#0;
   S711A_WELD_BUFF_DATA8.RBT8_BT_CODE_NO := W#16#0;
   S711A_WELD_BUFF_DATA8.RBT8_WELD_COUNT := W#16#0;
   S711A_WELD_BUFF_DATA8.RBT9_BT_CODE_NO := W#16#0;
   S711A_WELD_BUFF_DATA8.RBT9_WELD_COUNT := W#16#0;
   S711A_WELD_BUFF_DATA8.RBT10_BT_CODE_NO := W#16#0;
   S711A_WELD_BUFF_DATA8.RBT10_WELD_COUNT := W#16#0;
   S711A_WELD_BUFF_DATA8.RBT11_BT_CODE_NO := W#16#0;
   S711A_WELD_BUFF_DATA8.RBT11_WELD_COUNT := W#16#0;
   S711A_WELD_BUFF_DATA8.RBT12_BT_CODE_NO := W#16#0;
   S711A_WELD_BUFF_DATA8.RBT12_WELD_COUNT := W#16#0;
   S711A_WELD_BUFF_DATA8.RBT13_BT_CODE_NO := W#16#0;
   S711A_WELD_BUFF_DATA8.RBT13_WELD_COUNT := W#16#0;
   S711A_WELD_BUFF_DATA8.RBT14_BT_CODE_NO := W#16#0;
   S711A_WELD_BUFF_DATA8.RBT14_WELD_COUNT := W#16#0;
   S711A_WELD_BUFF_DATA8.RBT15_BT_CODE_NO := W#16#0;
   S711A_WELD_BUFF_DATA8.RBT15_WELD_COUNT := W#16#0;
   S711A_WELD_BUFF_DATA8.RBT16_BT_CODE_NO := W#16#0;
   S711A_WELD_BUFF_DATA8.RBT16_WELD_COUNT := W#16#0;
   S711A_WELD_BUFF_DATA8.RBT17_BT_CODE_NO := W#16#0;
   S711A_WELD_BUFF_DATA8.RBT17_WELD_COUNT := W#16#0;
   S711A_WELD_BUFF_DATA8.RBT18_BT_CODE_NO := W#16#0;
   S711A_WELD_BUFF_DATA8.RBT18_WELD_COUNT := W#16#0;
   S711A_WELD_BUFF_DATA8.RBT19_BT_CODE_NO := W#16#0;
   S711A_WELD_BUFF_DATA8.RBT19_WELD_COUNT := W#16#0;
   S711A_WELD_BUFF_DATA8.RBT20_BT_CODE_NO := W#16#0;
   S711A_WELD_BUFF_DATA8.RBT20_WELD_COUNT := W#16#0;
   S711A_WELD_BUFF_DATA8.RBT21_BT_CODE_NO := W#16#0;
   S711A_WELD_BUFF_DATA8.RBT21_WELD_COUNT := W#16#0;
   S711A_WELD_BUFF_DATA8.RBT22_BT_CODE_NO := W#16#0;
   S711A_WELD_BUFF_DATA8.RBT22_WELD_COUNT := W#16#0;
   S711A_WELD_BUFF_DATA8.RBT23_BT_CODE_NO := W#16#0;
   S711A_WELD_BUFF_DATA8.RBT23_WELD_COUNT := W#16#0;
   S711A_WELD_BUFF_DATA8.RBT24_BT_CODE_NO := W#16#0;
   S711A_WELD_BUFF_DATA8.RBT24_WELD_COUNT := W#16#0;
   S711A_WELD_BUFF_DATA8.WELD_DETERMINES_RESULT := W#16#0;
   S711A_WELD_BUFF_DATA8.WELD_CHECK_SUM := W#16#0;
   S711A_WELD_BUFF_DATA8.SPARE1 := W#16#0;
   S711A_WELD_BUFF_DATA9.STATION_MAIN := W#16#0;
   S711A_WELD_BUFF_DATA9.DISTINCTION_LH_RH := W#16#0;
   S711A_WELD_BUFF_DATA9.STAION_NUMBER := W#16#0;
   S711A_WELD_BUFF_DATA9.VIN_NUMBER1 := W#16#0;
   S711A_WELD_BUFF_DATA9.VIN_NUMBER2 := W#16#0;
   S711A_WELD_BUFF_DATA9.VIN_NUMBER3 := W#16#0;
   S711A_WELD_BUFF_DATA9.VIN_NUMBER4 := W#16#0;
   S711A_WELD_BUFF_DATA9.SEQ_NUMBER1 := W#16#0;
   S711A_WELD_BUFF_DATA9.SEQ_NUMBER2 := W#16#0;
   S711A_WELD_BUFF_DATA9.RBT1_BT_CODE_NO := W#16#0;
   S711A_WELD_BUFF_DATA9.RBT1_WELD_COUNT := W#16#0;
   S711A_WELD_BUFF_DATA9.RBT2_BT_CODE_NO := W#16#0;
   S711A_WELD_BUFF_DATA9.RBT2_WELD_COUNT := W#16#0;
   S711A_WELD_BUFF_DATA9.RBT3_BT_CODE_NO := W#16#0;
   S711A_WELD_BUFF_DATA9.RBT3_WELD_COUNT := W#16#0;
   S711A_WELD_BUFF_DATA9.RBT4_BT_CODE_NO := W#16#0;
   S711A_WELD_BUFF_DATA9.RBT4_WELD_COUNT := W#16#0;
   S711A_WELD_BUFF_DATA9.RBT5_BT_CODE_NO := W#16#0;
   S711A_WELD_BUFF_DATA9.RBT5_WELD_COUNT := W#16#0;
   S711A_WELD_BUFF_DATA9.RBT6_BT_CODE_NO := W#16#0;
   S711A_WELD_BUFF_DATA9.RBT6_WELD_COUNT := W#16#0;
   S711A_WELD_BUFF_DATA9.RBT7_BT_CODE_NO := W#16#0;
   S711A_WELD_BUFF_DATA9.RBT7_WELD_COUNT := W#16#0;
   S711A_WELD_BUFF_DATA9.RBT8_BT_CODE_NO := W#16#0;
   S711A_WELD_BUFF_DATA9.RBT8_WELD_COUNT := W#16#0;
   S711A_WELD_BUFF_DATA9.RBT9_BT_CODE_NO := W#16#0;
   S711A_WELD_BUFF_DATA9.RBT9_WELD_COUNT := W#16#0;
   S711A_WELD_BUFF_DATA9.RBT10_BT_CODE_NO := W#16#0;
   S711A_WELD_BUFF_DATA9.RBT10_WELD_COUNT := W#16#0;
   S711A_WELD_BUFF_DATA9.RBT11_BT_CODE_NO := W#16#0;
   S711A_WELD_BUFF_DATA9.RBT11_WELD_COUNT := W#16#0;
   S711A_WELD_BUFF_DATA9.RBT12_BT_CODE_NO := W#16#0;
   S711A_WELD_BUFF_DATA9.RBT12_WELD_COUNT := W#16#0;
   S711A_WELD_BUFF_DATA9.RBT13_BT_CODE_NO := W#16#0;
   S711A_WELD_BUFF_DATA9.RBT13_WELD_COUNT := W#16#0;
   S711A_WELD_BUFF_DATA9.RBT14_BT_CODE_NO := W#16#0;
   S711A_WELD_BUFF_DATA9.RBT14_WELD_COUNT := W#16#0;
   S711A_WELD_BUFF_DATA9.RBT15_BT_CODE_NO := W#16#0;
   S711A_WELD_BUFF_DATA9.RBT15_WELD_COUNT := W#16#0;
   S711A_WELD_BUFF_DATA9.RBT16_BT_CODE_NO := W#16#0;
   S711A_WELD_BUFF_DATA9.RBT16_WELD_COUNT := W#16#0;
   S711A_WELD_BUFF_DATA9.RBT17_BT_CODE_NO := W#16#0;
   S711A_WELD_BUFF_DATA9.RBT17_WELD_COUNT := W#16#0;
   S711A_WELD_BUFF_DATA9.RBT18_BT_CODE_NO := W#16#0;
   S711A_WELD_BUFF_DATA9.RBT18_WELD_COUNT := W#16#0;
   S711A_WELD_BUFF_DATA9.RBT19_BT_CODE_NO := W#16#0;
   S711A_WELD_BUFF_DATA9.RBT19_WELD_COUNT := W#16#0;
   S711A_WELD_BUFF_DATA9.RBT20_BT_CODE_NO := W#16#0;
   S711A_WELD_BUFF_DATA9.RBT20_WELD_COUNT := W#16#0;
   S711A_WELD_BUFF_DATA9.RBT21_BT_CODE_NO := W#16#0;
   S711A_WELD_BUFF_DATA9.RBT21_WELD_COUNT := W#16#0;
   S711A_WELD_BUFF_DATA9.RBT22_BT_CODE_NO := W#16#0;
   S711A_WELD_BUFF_DATA9.RBT22_WELD_COUNT := W#16#0;
   S711A_WELD_BUFF_DATA9.RBT23_BT_CODE_NO := W#16#0;
   S711A_WELD_BUFF_DATA9.RBT23_WELD_COUNT := W#16#0;
   S711A_WELD_BUFF_DATA9.RBT24_BT_CODE_NO := W#16#0;
   S711A_WELD_BUFF_DATA9.RBT24_WELD_COUNT := W#16#0;
   S711A_WELD_BUFF_DATA9.WELD_DETERMINES_RESULT := W#16#0;
   S711A_WELD_BUFF_DATA9.WELD_CHECK_SUM := W#16#0;
   S711A_WELD_BUFF_DATA9.SPARE1 := W#16#0;
   S711A_WELD_BUFF_DATA10.STATION_MAIN := W#16#0;
   S711A_WELD_BUFF_DATA10.DISTINCTION_LH_RH := W#16#0;
   S711A_WELD_BUFF_DATA10.STAION_NUMBER := W#16#0;
   S711A_WELD_BUFF_DATA10.VIN_NUMBER1 := W#16#0;
   S711A_WELD_BUFF_DATA10.VIN_NUMBER2 := W#16#0;
   S711A_WELD_BUFF_DATA10.VIN_NUMBER3 := W#16#0;
   S711A_WELD_BUFF_DATA10.VIN_NUMBER4 := W#16#0;
   S711A_WELD_BUFF_DATA10.SEQ_NUMBER1 := W#16#0;
   S711A_WELD_BUFF_DATA10.SEQ_NUMBER2 := W#16#0;
   S711A_WELD_BUFF_DATA10.RBT1_BT_CODE_NO := W#16#0;
   S711A_WELD_BUFF_DATA10.RBT1_WELD_COUNT := W#16#0;
   S711A_WELD_BUFF_DATA10.RBT2_BT_CODE_NO := W#16#0;
   S711A_WELD_BUFF_DATA10.RBT2_WELD_COUNT := W#16#0;
   S711A_WELD_BUFF_DATA10.RBT3_BT_CODE_NO := W#16#0;
   S711A_WELD_BUFF_DATA10.RBT3_WELD_COUNT := W#16#0;
   S711A_WELD_BUFF_DATA10.RBT4_BT_CODE_NO := W#16#0;
   S711A_WELD_BUFF_DATA10.RBT4_WELD_COUNT := W#16#0;
   S711A_WELD_BUFF_DATA10.RBT5_BT_CODE_NO := W#16#0;
   S711A_WELD_BUFF_DATA10.RBT5_WELD_COUNT := W#16#0;
   S711A_WELD_BUFF_DATA10.RBT6_BT_CODE_NO := W#16#0;
   S711A_WELD_BUFF_DATA10.RBT6_WELD_COUNT := W#16#0;
   S711A_WELD_BUFF_DATA10.RBT7_BT_CODE_NO := W#16#0;
   S711A_WELD_BUFF_DATA10.RBT7_WELD_COUNT := W#16#0;
   S711A_WELD_BUFF_DATA10.RBT8_BT_CODE_NO := W#16#0;
   S711A_WELD_BUFF_DATA10.RBT8_WELD_COUNT := W#16#0;
   S711A_WELD_BUFF_DATA10.RBT9_BT_CODE_NO := W#16#0;
   S711A_WELD_BUFF_DATA10.RBT9_WELD_COUNT := W#16#0;
   S711A_WELD_BUFF_DATA10.RBT10_BT_CODE_NO := W#16#0;
   S711A_WELD_BUFF_DATA10.RBT10_WELD_COUNT := W#16#0;
   S711A_WELD_BUFF_DATA10.RBT11_BT_CODE_NO := W#16#0;
   S711A_WELD_BUFF_DATA10.RBT11_WELD_COUNT := W#16#0;
   S711A_WELD_BUFF_DATA10.RBT12_BT_CODE_NO := W#16#0;
   S711A_WELD_BUFF_DATA10.RBT12_WELD_COUNT := W#16#0;
   S711A_WELD_BUFF_DATA10.RBT13_BT_CODE_NO := W#16#0;
   S711A_WELD_BUFF_DATA10.RBT13_WELD_COUNT := W#16#0;
   S711A_WELD_BUFF_DATA10.RBT14_BT_CODE_NO := W#16#0;
   S711A_WELD_BUFF_DATA10.RBT14_WELD_COUNT := W#16#0;
   S711A_WELD_BUFF_DATA10.RBT15_BT_CODE_NO := W#16#0;
   S711A_WELD_BUFF_DATA10.RBT15_WELD_COUNT := W#16#0;
   S711A_WELD_BUFF_DATA10.RBT16_BT_CODE_NO := W#16#0;
   S711A_WELD_BUFF_DATA10.RBT16_WELD_COUNT := W#16#0;
   S711A_WELD_BUFF_DATA10.RBT17_BT_CODE_NO := W#16#0;
   S711A_WELD_BUFF_DATA10.RBT17_WELD_COUNT := W#16#0;
   S711A_WELD_BUFF_DATA10.RBT18_BT_CODE_NO := W#16#0;
   S711A_WELD_BUFF_DATA10.RBT18_WELD_COUNT := W#16#0;
   S711A_WELD_BUFF_DATA10.RBT19_BT_CODE_NO := W#16#0;
   S711A_WELD_BUFF_DATA10.RBT19_WELD_COUNT := W#16#0;
   S711A_WELD_BUFF_DATA10.RBT20_BT_CODE_NO := W#16#0;
   S711A_WELD_BUFF_DATA10.RBT20_WELD_COUNT := W#16#0;
   S711A_WELD_BUFF_DATA10.RBT21_BT_CODE_NO := W#16#0;
   S711A_WELD_BUFF_DATA10.RBT21_WELD_COUNT := W#16#0;
   S711A_WELD_BUFF_DATA10.RBT22_BT_CODE_NO := W#16#0;
   S711A_WELD_BUFF_DATA10.RBT22_WELD_COUNT := W#16#0;
   S711A_WELD_BUFF_DATA10.RBT23_BT_CODE_NO := W#16#0;
   S711A_WELD_BUFF_DATA10.RBT23_WELD_COUNT := W#16#0;
   S711A_WELD_BUFF_DATA10.RBT24_BT_CODE_NO := W#16#0;
   S711A_WELD_BUFF_DATA10.RBT24_WELD_COUNT := W#16#0;
   S711A_WELD_BUFF_DATA10.WELD_DETERMINES_RESULT := W#16#0;
   S711A_WELD_BUFF_DATA10.WELD_CHECK_SUM := W#16#0;
   S711A_WELD_BUFF_DATA10.SPARE1 := W#16#0;
   S711_WELD_BUFF_DATA1.STATION_MAIN := W#16#0;
   S711_WELD_BUFF_DATA1.DISTINCTION_LH_RH := W#16#0;
   S711_WELD_BUFF_DATA1.STAION_NUMBER := W#16#0;
   S711_WELD_BUFF_DATA1.VIN_NUMBER1 := W#16#0;
   S711_WELD_BUFF_DATA1.VIN_NUMBER2 := W#16#0;
   S711_WELD_BUFF_DATA1.VIN_NUMBER3 := W#16#0;
   S711_WELD_BUFF_DATA1.VIN_NUMBER4 := W#16#0;
   S711_WELD_BUFF_DATA1.SEQ_NUMBER1 := W#16#0;
   S711_WELD_BUFF_DATA1.SEQ_NUMBER2 := W#16#0;
   S711_WELD_BUFF_DATA1.RBT1_BT_CODE_NO := W#16#0;
   S711_WELD_BUFF_DATA1.RBT1_WELD_COUNT := W#16#0;
   S711_WELD_BUFF_DATA1.RBT2_BT_CODE_NO := W#16#0;
   S711_WELD_BUFF_DATA1.RBT2_WELD_COUNT := W#16#0;
   S711_WELD_BUFF_DATA1.RBT3_BT_CODE_NO := W#16#0;
   S711_WELD_BUFF_DATA1.RBT3_WELD_COUNT := W#16#0;
   S711_WELD_BUFF_DATA1.RBT4_BT_CODE_NO := W#16#0;
   S711_WELD_BUFF_DATA1.RBT4_WELD_COUNT := W#16#0;
   S711_WELD_BUFF_DATA1.RBT5_BT_CODE_NO := W#16#0;
   S711_WELD_BUFF_DATA1.RBT5_WELD_COUNT := W#16#0;
   S711_WELD_BUFF_DATA1.RBT6_BT_CODE_NO := W#16#0;
   S711_WELD_BUFF_DATA1.RBT6_WELD_COUNT := W#16#0;
   S711_WELD_BUFF_DATA1.RBT7_BT_CODE_NO := W#16#0;
   S711_WELD_BUFF_DATA1.RBT7_WELD_COUNT := W#16#0;
   S711_WELD_BUFF_DATA1.RBT8_BT_CODE_NO := W#16#0;
   S711_WELD_BUFF_DATA1.RBT8_WELD_COUNT := W#16#0;
   S711_WELD_BUFF_DATA1.RBT9_BT_CODE_NO := W#16#0;
   S711_WELD_BUFF_DATA1.RBT9_WELD_COUNT := W#16#0;
   S711_WELD_BUFF_DATA1.RBT10_BT_CODE_NO := W#16#0;
   S711_WELD_BUFF_DATA1.RBT10_WELD_COUNT := W#16#0;
   S711_WELD_BUFF_DATA1.RBT11_BT_CODE_NO := W#16#0;
   S711_WELD_BUFF_DATA1.RBT11_WELD_COUNT := W#16#0;
   S711_WELD_BUFF_DATA1.RBT12_BT_CODE_NO := W#16#0;
   S711_WELD_BUFF_DATA1.RBT12_WELD_COUNT := W#16#0;
   S711_WELD_BUFF_DATA1.RBT13_BT_CODE_NO := W#16#0;
   S711_WELD_BUFF_DATA1.RBT13_WELD_COUNT := W#16#0;
   S711_WELD_BUFF_DATA1.RBT14_BT_CODE_NO := W#16#0;
   S711_WELD_BUFF_DATA1.RBT14_WELD_COUNT := W#16#0;
   S711_WELD_BUFF_DATA1.RBT15_BT_CODE_NO := W#16#0;
   S711_WELD_BUFF_DATA1.RBT15_WELD_COUNT := W#16#0;
   S711_WELD_BUFF_DATA1.RBT16_BT_CODE_NO := W#16#0;
   S711_WELD_BUFF_DATA1.RBT16_WELD_COUNT := W#16#0;
   S711_WELD_BUFF_DATA1.RBT17_BT_CODE_NO := W#16#0;
   S711_WELD_BUFF_DATA1.RBT17_WELD_COUNT := W#16#0;
   S711_WELD_BUFF_DATA1.RBT18_BT_CODE_NO := W#16#0;
   S711_WELD_BUFF_DATA1.RBT18_WELD_COUNT := W#16#0;
   S711_WELD_BUFF_DATA1.RBT19_BT_CODE_NO := W#16#0;
   S711_WELD_BUFF_DATA1.RBT19_WELD_COUNT := W#16#0;
   S711_WELD_BUFF_DATA1.RBT20_BT_CODE_NO := W#16#0;
   S711_WELD_BUFF_DATA1.RBT20_WELD_COUNT := W#16#0;
   S711_WELD_BUFF_DATA1.RBT21_BT_CODE_NO := W#16#0;
   S711_WELD_BUFF_DATA1.RBT21_WELD_COUNT := W#16#0;
   S711_WELD_BUFF_DATA1.RBT22_BT_CODE_NO := W#16#0;
   S711_WELD_BUFF_DATA1.RBT22_WELD_COUNT := W#16#0;
   S711_WELD_BUFF_DATA1.RBT23_BT_CODE_NO := W#16#0;
   S711_WELD_BUFF_DATA1.RBT23_WELD_COUNT := W#16#0;
   S711_WELD_BUFF_DATA1.RBT24_BT_CODE_NO := W#16#0;
   S711_WELD_BUFF_DATA1.RBT24_WELD_COUNT := W#16#0;
   S711_WELD_BUFF_DATA1.WELD_DETERMINES_RESULT := W#16#0;
   S711_WELD_BUFF_DATA1.WELD_CHECK_SUM := W#16#0;
   S711_WELD_BUFF_DATA1.SPARE1 := W#16#0;
   S711_WELD_BUFF_DATA2.STATION_MAIN := W#16#0;
   S711_WELD_BUFF_DATA2.DISTINCTION_LH_RH := W#16#0;
   S711_WELD_BUFF_DATA2.STAION_NUMBER := W#16#0;
   S711_WELD_BUFF_DATA2.VIN_NUMBER1 := W#16#0;
   S711_WELD_BUFF_DATA2.VIN_NUMBER2 := W#16#0;
   S711_WELD_BUFF_DATA2.VIN_NUMBER3 := W#16#0;
   S711_WELD_BUFF_DATA2.VIN_NUMBER4 := W#16#0;
   S711_WELD_BUFF_DATA2.SEQ_NUMBER1 := W#16#0;
   S711_WELD_BUFF_DATA2.SEQ_NUMBER2 := W#16#0;
   S711_WELD_BUFF_DATA2.RBT1_BT_CODE_NO := W#16#0;
   S711_WELD_BUFF_DATA2.RBT1_WELD_COUNT := W#16#0;
   S711_WELD_BUFF_DATA2.RBT2_BT_CODE_NO := W#16#0;
   S711_WELD_BUFF_DATA2.RBT2_WELD_COUNT := W#16#0;
   S711_WELD_BUFF_DATA2.RBT3_BT_CODE_NO := W#16#0;
   S711_WELD_BUFF_DATA2.RBT3_WELD_COUNT := W#16#0;
   S711_WELD_BUFF_DATA2.RBT4_BT_CODE_NO := W#16#0;
   S711_WELD_BUFF_DATA2.RBT4_WELD_COUNT := W#16#0;
   S711_WELD_BUFF_DATA2.RBT5_BT_CODE_NO := W#16#0;
   S711_WELD_BUFF_DATA2.RBT5_WELD_COUNT := W#16#0;
   S711_WELD_BUFF_DATA2.RBT6_BT_CODE_NO := W#16#0;
   S711_WELD_BUFF_DATA2.RBT6_WELD_COUNT := W#16#0;
   S711_WELD_BUFF_DATA2.RBT7_BT_CODE_NO := W#16#0;
   S711_WELD_BUFF_DATA2.RBT7_WELD_COUNT := W#16#0;
   S711_WELD_BUFF_DATA2.RBT8_BT_CODE_NO := W#16#0;
   S711_WELD_BUFF_DATA2.RBT8_WELD_COUNT := W#16#0;
   S711_WELD_BUFF_DATA2.RBT9_BT_CODE_NO := W#16#0;
   S711_WELD_BUFF_DATA2.RBT9_WELD_COUNT := W#16#0;
   S711_WELD_BUFF_DATA2.RBT10_BT_CODE_NO := W#16#0;
   S711_WELD_BUFF_DATA2.RBT10_WELD_COUNT := W#16#0;
   S711_WELD_BUFF_DATA2.RBT11_BT_CODE_NO := W#16#0;
   S711_WELD_BUFF_DATA2.RBT11_WELD_COUNT := W#16#0;
   S711_WELD_BUFF_DATA2.RBT12_BT_CODE_NO := W#16#0;
   S711_WELD_BUFF_DATA2.RBT12_WELD_COUNT := W#16#0;
   S711_WELD_BUFF_DATA2.RBT13_BT_CODE_NO := W#16#0;
   S711_WELD_BUFF_DATA2.RBT13_WELD_COUNT := W#16#0;
   S711_WELD_BUFF_DATA2.RBT14_BT_CODE_NO := W#16#0;
   S711_WELD_BUFF_DATA2.RBT14_WELD_COUNT := W#16#0;
   S711_WELD_BUFF_DATA2.RBT15_BT_CODE_NO := W#16#0;
   S711_WELD_BUFF_DATA2.RBT15_WELD_COUNT := W#16#0;
   S711_WELD_BUFF_DATA2.RBT16_BT_CODE_NO := W#16#0;
   S711_WELD_BUFF_DATA2.RBT16_WELD_COUNT := W#16#0;
   S711_WELD_BUFF_DATA2.RBT17_BT_CODE_NO := W#16#0;
   S711_WELD_BUFF_DATA2.RBT17_WELD_COUNT := W#16#0;
   S711_WELD_BUFF_DATA2.RBT18_BT_CODE_NO := W#16#0;
   S711_WELD_BUFF_DATA2.RBT18_WELD_COUNT := W#16#0;
   S711_WELD_BUFF_DATA2.RBT19_BT_CODE_NO := W#16#0;
   S711_WELD_BUFF_DATA2.RBT19_WELD_COUNT := W#16#0;
   S711_WELD_BUFF_DATA2.RBT20_BT_CODE_NO := W#16#0;
   S711_WELD_BUFF_DATA2.RBT20_WELD_COUNT := W#16#0;
   S711_WELD_BUFF_DATA2.RBT21_BT_CODE_NO := W#16#0;
   S711_WELD_BUFF_DATA2.RBT21_WELD_COUNT := W#16#0;
   S711_WELD_BUFF_DATA2.RBT22_BT_CODE_NO := W#16#0;
   S711_WELD_BUFF_DATA2.RBT22_WELD_COUNT := W#16#0;
   S711_WELD_BUFF_DATA2.RBT23_BT_CODE_NO := W#16#0;
   S711_WELD_BUFF_DATA2.RBT23_WELD_COUNT := W#16#0;
   S711_WELD_BUFF_DATA2.RBT24_BT_CODE_NO := W#16#0;
   S711_WELD_BUFF_DATA2.RBT24_WELD_COUNT := W#16#0;
   S711_WELD_BUFF_DATA2.WELD_DETERMINES_RESULT := W#16#0;
   S711_WELD_BUFF_DATA2.WELD_CHECK_SUM := W#16#0;
   S711_WELD_BUFF_DATA2.SPARE1 := W#16#0;
   S711_WELD_BUFF_DATA3.STATION_MAIN := W#16#0;
   S711_WELD_BUFF_DATA3.DISTINCTION_LH_RH := W#16#0;
   S711_WELD_BUFF_DATA3.STAION_NUMBER := W#16#0;
   S711_WELD_BUFF_DATA3.VIN_NUMBER1 := W#16#0;
   S711_WELD_BUFF_DATA3.VIN_NUMBER2 := W#16#0;
   S711_WELD_BUFF_DATA3.VIN_NUMBER3 := W#16#0;
   S711_WELD_BUFF_DATA3.VIN_NUMBER4 := W#16#0;
   S711_WELD_BUFF_DATA3.SEQ_NUMBER1 := W#16#0;
   S711_WELD_BUFF_DATA3.SEQ_NUMBER2 := W#16#0;
   S711_WELD_BUFF_DATA3.RBT1_BT_CODE_NO := W#16#0;
   S711_WELD_BUFF_DATA3.RBT1_WELD_COUNT := W#16#0;
   S711_WELD_BUFF_DATA3.RBT2_BT_CODE_NO := W#16#0;
   S711_WELD_BUFF_DATA3.RBT2_WELD_COUNT := W#16#0;
   S711_WELD_BUFF_DATA3.RBT3_BT_CODE_NO := W#16#0;
   S711_WELD_BUFF_DATA3.RBT3_WELD_COUNT := W#16#0;
   S711_WELD_BUFF_DATA3.RBT4_BT_CODE_NO := W#16#0;
   S711_WELD_BUFF_DATA3.RBT4_WELD_COUNT := W#16#0;
   S711_WELD_BUFF_DATA3.RBT5_BT_CODE_NO := W#16#0;
   S711_WELD_BUFF_DATA3.RBT5_WELD_COUNT := W#16#0;
   S711_WELD_BUFF_DATA3.RBT6_BT_CODE_NO := W#16#0;
   S711_WELD_BUFF_DATA3.RBT6_WELD_COUNT := W#16#0;
   S711_WELD_BUFF_DATA3.RBT7_BT_CODE_NO := W#16#0;
   S711_WELD_BUFF_DATA3.RBT7_WELD_COUNT := W#16#0;
   S711_WELD_BUFF_DATA3.RBT8_BT_CODE_NO := W#16#0;
   S711_WELD_BUFF_DATA3.RBT8_WELD_COUNT := W#16#0;
   S711_WELD_BUFF_DATA3.RBT9_BT_CODE_NO := W#16#0;
   S711_WELD_BUFF_DATA3.RBT9_WELD_COUNT := W#16#0;
   S711_WELD_BUFF_DATA3.RBT10_BT_CODE_NO := W#16#0;
   S711_WELD_BUFF_DATA3.RBT10_WELD_COUNT := W#16#0;
   S711_WELD_BUFF_DATA3.RBT11_BT_CODE_NO := W#16#0;
   S711_WELD_BUFF_DATA3.RBT11_WELD_COUNT := W#16#0;
   S711_WELD_BUFF_DATA3.RBT12_BT_CODE_NO := W#16#0;
   S711_WELD_BUFF_DATA3.RBT12_WELD_COUNT := W#16#0;
   S711_WELD_BUFF_DATA3.RBT13_BT_CODE_NO := W#16#0;
   S711_WELD_BUFF_DATA3.RBT13_WELD_COUNT := W#16#0;
   S711_WELD_BUFF_DATA3.RBT14_BT_CODE_NO := W#16#0;
   S711_WELD_BUFF_DATA3.RBT14_WELD_COUNT := W#16#0;
   S711_WELD_BUFF_DATA3.RBT15_BT_CODE_NO := W#16#0;
   S711_WELD_BUFF_DATA3.RBT15_WELD_COUNT := W#16#0;
   S711_WELD_BUFF_DATA3.RBT16_BT_CODE_NO := W#16#0;
   S711_WELD_BUFF_DATA3.RBT16_WELD_COUNT := W#16#0;
   S711_WELD_BUFF_DATA3.RBT17_BT_CODE_NO := W#16#0;
   S711_WELD_BUFF_DATA3.RBT17_WELD_COUNT := W#16#0;
   S711_WELD_BUFF_DATA3.RBT18_BT_CODE_NO := W#16#0;
   S711_WELD_BUFF_DATA3.RBT18_WELD_COUNT := W#16#0;
   S711_WELD_BUFF_DATA3.RBT19_BT_CODE_NO := W#16#0;
   S711_WELD_BUFF_DATA3.RBT19_WELD_COUNT := W#16#0;
   S711_WELD_BUFF_DATA3.RBT20_BT_CODE_NO := W#16#0;
   S711_WELD_BUFF_DATA3.RBT20_WELD_COUNT := W#16#0;
   S711_WELD_BUFF_DATA3.RBT21_BT_CODE_NO := W#16#0;
   S711_WELD_BUFF_DATA3.RBT21_WELD_COUNT := W#16#0;
   S711_WELD_BUFF_DATA3.RBT22_BT_CODE_NO := W#16#0;
   S711_WELD_BUFF_DATA3.RBT22_WELD_COUNT := W#16#0;
   S711_WELD_BUFF_DATA3.RBT23_BT_CODE_NO := W#16#0;
   S711_WELD_BUFF_DATA3.RBT23_WELD_COUNT := W#16#0;
   S711_WELD_BUFF_DATA3.RBT24_BT_CODE_NO := W#16#0;
   S711_WELD_BUFF_DATA3.RBT24_WELD_COUNT := W#16#0;
   S711_WELD_BUFF_DATA3.WELD_DETERMINES_RESULT := W#16#0;
   S711_WELD_BUFF_DATA3.WELD_CHECK_SUM := W#16#0;
   S711_WELD_BUFF_DATA3.SPARE1 := W#16#0;
   S711_WELD_BUFF_DATA4.STATION_MAIN := W#16#0;
   S711_WELD_BUFF_DATA4.DISTINCTION_LH_RH := W#16#0;
   S711_WELD_BUFF_DATA4.STAION_NUMBER := W#16#0;
   S711_WELD_BUFF_DATA4.VIN_NUMBER1 := W#16#0;
   S711_WELD_BUFF_DATA4.VIN_NUMBER2 := W#16#0;
   S711_WELD_BUFF_DATA4.VIN_NUMBER3 := W#16#0;
   S711_WELD_BUFF_DATA4.VIN_NUMBER4 := W#16#0;
   S711_WELD_BUFF_DATA4.SEQ_NUMBER1 := W#16#0;
   S711_WELD_BUFF_DATA4.SEQ_NUMBER2 := W#16#0;
   S711_WELD_BUFF_DATA4.RBT1_BT_CODE_NO := W#16#0;
   S711_WELD_BUFF_DATA4.RBT1_WELD_COUNT := W#16#0;
   S711_WELD_BUFF_DATA4.RBT2_BT_CODE_NO := W#16#0;
   S711_WELD_BUFF_DATA4.RBT2_WELD_COUNT := W#16#0;
   S711_WELD_BUFF_DATA4.RBT3_BT_CODE_NO := W#16#0;
   S711_WELD_BUFF_DATA4.RBT3_WELD_COUNT := W#16#0;
   S711_WELD_BUFF_DATA4.RBT4_BT_CODE_NO := W#16#0;
   S711_WELD_BUFF_DATA4.RBT4_WELD_COUNT := W#16#0;
   S711_WELD_BUFF_DATA4.RBT5_BT_CODE_NO := W#16#0;
   S711_WELD_BUFF_DATA4.RBT5_WELD_COUNT := W#16#0;
   S711_WELD_BUFF_DATA4.RBT6_BT_CODE_NO := W#16#0;
   S711_WELD_BUFF_DATA4.RBT6_WELD_COUNT := W#16#0;
   S711_WELD_BUFF_DATA4.RBT7_BT_CODE_NO := W#16#0;
   S711_WELD_BUFF_DATA4.RBT7_WELD_COUNT := W#16#0;
   S711_WELD_BUFF_DATA4.RBT8_BT_CODE_NO := W#16#0;
   S711_WELD_BUFF_DATA4.RBT8_WELD_COUNT := W#16#0;
   S711_WELD_BUFF_DATA4.RBT9_BT_CODE_NO := W#16#0;
   S711_WELD_BUFF_DATA4.RBT9_WELD_COUNT := W#16#0;
   S711_WELD_BUFF_DATA4.RBT10_BT_CODE_NO := W#16#0;
   S711_WELD_BUFF_DATA4.RBT10_WELD_COUNT := W#16#0;
   S711_WELD_BUFF_DATA4.RBT11_BT_CODE_NO := W#16#0;
   S711_WELD_BUFF_DATA4.RBT11_WELD_COUNT := W#16#0;
   S711_WELD_BUFF_DATA4.RBT12_BT_CODE_NO := W#16#0;
   S711_WELD_BUFF_DATA4.RBT12_WELD_COUNT := W#16#0;
   S711_WELD_BUFF_DATA4.RBT13_BT_CODE_NO := W#16#0;
   S711_WELD_BUFF_DATA4.RBT13_WELD_COUNT := W#16#0;
   S711_WELD_BUFF_DATA4.RBT14_BT_CODE_NO := W#16#0;
   S711_WELD_BUFF_DATA4.RBT14_WELD_COUNT := W#16#0;
   S711_WELD_BUFF_DATA4.RBT15_BT_CODE_NO := W#16#0;
   S711_WELD_BUFF_DATA4.RBT15_WELD_COUNT := W#16#0;
   S711_WELD_BUFF_DATA4.RBT16_BT_CODE_NO := W#16#0;
   S711_WELD_BUFF_DATA4.RBT16_WELD_COUNT := W#16#0;
   S711_WELD_BUFF_DATA4.RBT17_BT_CODE_NO := W#16#0;
   S711_WELD_BUFF_DATA4.RBT17_WELD_COUNT := W#16#0;
   S711_WELD_BUFF_DATA4.RBT18_BT_CODE_NO := W#16#0;
   S711_WELD_BUFF_DATA4.RBT18_WELD_COUNT := W#16#0;
   S711_WELD_BUFF_DATA4.RBT19_BT_CODE_NO := W#16#0;
   S711_WELD_BUFF_DATA4.RBT19_WELD_COUNT := W#16#0;
   S711_WELD_BUFF_DATA4.RBT20_BT_CODE_NO := W#16#0;
   S711_WELD_BUFF_DATA4.RBT20_WELD_COUNT := W#16#0;
   S711_WELD_BUFF_DATA4.RBT21_BT_CODE_NO := W#16#0;
   S711_WELD_BUFF_DATA4.RBT21_WELD_COUNT := W#16#0;
   S711_WELD_BUFF_DATA4.RBT22_BT_CODE_NO := W#16#0;
   S711_WELD_BUFF_DATA4.RBT22_WELD_COUNT := W#16#0;
   S711_WELD_BUFF_DATA4.RBT23_BT_CODE_NO := W#16#0;
   S711_WELD_BUFF_DATA4.RBT23_WELD_COUNT := W#16#0;
   S711_WELD_BUFF_DATA4.RBT24_BT_CODE_NO := W#16#0;
   S711_WELD_BUFF_DATA4.RBT24_WELD_COUNT := W#16#0;
   S711_WELD_BUFF_DATA4.WELD_DETERMINES_RESULT := W#16#0;
   S711_WELD_BUFF_DATA4.WELD_CHECK_SUM := W#16#0;
   S711_WELD_BUFF_DATA4.SPARE1 := W#16#0;
   S711_WELD_BUFF_DATA5.STATION_MAIN := W#16#0;
   S711_WELD_BUFF_DATA5.DISTINCTION_LH_RH := W#16#0;
   S711_WELD_BUFF_DATA5.STAION_NUMBER := W#16#0;
   S711_WELD_BUFF_DATA5.VIN_NUMBER1 := W#16#0;
   S711_WELD_BUFF_DATA5.VIN_NUMBER2 := W#16#0;
   S711_WELD_BUFF_DATA5.VIN_NUMBER3 := W#16#0;
   S711_WELD_BUFF_DATA5.VIN_NUMBER4 := W#16#0;
   S711_WELD_BUFF_DATA5.SEQ_NUMBER1 := W#16#0;
   S711_WELD_BUFF_DATA5.SEQ_NUMBER2 := W#16#0;
   S711_WELD_BUFF_DATA5.RBT1_BT_CODE_NO := W#16#0;
   S711_WELD_BUFF_DATA5.RBT1_WELD_COUNT := W#16#0;
   S711_WELD_BUFF_DATA5.RBT2_BT_CODE_NO := W#16#0;
   S711_WELD_BUFF_DATA5.RBT2_WELD_COUNT := W#16#0;
   S711_WELD_BUFF_DATA5.RBT3_BT_CODE_NO := W#16#0;
   S711_WELD_BUFF_DATA5.RBT3_WELD_COUNT := W#16#0;
   S711_WELD_BUFF_DATA5.RBT4_BT_CODE_NO := W#16#0;
   S711_WELD_BUFF_DATA5.RBT4_WELD_COUNT := W#16#0;
   S711_WELD_BUFF_DATA5.RBT5_BT_CODE_NO := W#16#0;
   S711_WELD_BUFF_DATA5.RBT5_WELD_COUNT := W#16#0;
   S711_WELD_BUFF_DATA5.RBT6_BT_CODE_NO := W#16#0;
   S711_WELD_BUFF_DATA5.RBT6_WELD_COUNT := W#16#0;
   S711_WELD_BUFF_DATA5.RBT7_BT_CODE_NO := W#16#0;
   S711_WELD_BUFF_DATA5.RBT7_WELD_COUNT := W#16#0;
   S711_WELD_BUFF_DATA5.RBT8_BT_CODE_NO := W#16#0;
   S711_WELD_BUFF_DATA5.RBT8_WELD_COUNT := W#16#0;
   S711_WELD_BUFF_DATA5.RBT9_BT_CODE_NO := W#16#0;
   S711_WELD_BUFF_DATA5.RBT9_WELD_COUNT := W#16#0;
   S711_WELD_BUFF_DATA5.RBT10_BT_CODE_NO := W#16#0;
   S711_WELD_BUFF_DATA5.RBT10_WELD_COUNT := W#16#0;
   S711_WELD_BUFF_DATA5.RBT11_BT_CODE_NO := W#16#0;
   S711_WELD_BUFF_DATA5.RBT11_WELD_COUNT := W#16#0;
   S711_WELD_BUFF_DATA5.RBT12_BT_CODE_NO := W#16#0;
   S711_WELD_BUFF_DATA5.RBT12_WELD_COUNT := W#16#0;
   S711_WELD_BUFF_DATA5.RBT13_BT_CODE_NO := W#16#0;
   S711_WELD_BUFF_DATA5.RBT13_WELD_COUNT := W#16#0;
   S711_WELD_BUFF_DATA5.RBT14_BT_CODE_NO := W#16#0;
   S711_WELD_BUFF_DATA5.RBT14_WELD_COUNT := W#16#0;
   S711_WELD_BUFF_DATA5.RBT15_BT_CODE_NO := W#16#0;
   S711_WELD_BUFF_DATA5.RBT15_WELD_COUNT := W#16#0;
   S711_WELD_BUFF_DATA5.RBT16_BT_CODE_NO := W#16#0;
   S711_WELD_BUFF_DATA5.RBT16_WELD_COUNT := W#16#0;
   S711_WELD_BUFF_DATA5.RBT17_BT_CODE_NO := W#16#0;
   S711_WELD_BUFF_DATA5.RBT17_WELD_COUNT := W#16#0;
   S711_WELD_BUFF_DATA5.RBT18_BT_CODE_NO := W#16#0;
   S711_WELD_BUFF_DATA5.RBT18_WELD_COUNT := W#16#0;
   S711_WELD_BUFF_DATA5.RBT19_BT_CODE_NO := W#16#0;
   S711_WELD_BUFF_DATA5.RBT19_WELD_COUNT := W#16#0;
   S711_WELD_BUFF_DATA5.RBT20_BT_CODE_NO := W#16#0;
   S711_WELD_BUFF_DATA5.RBT20_WELD_COUNT := W#16#0;
   S711_WELD_BUFF_DATA5.RBT21_BT_CODE_NO := W#16#0;
   S711_WELD_BUFF_DATA5.RBT21_WELD_COUNT := W#16#0;
   S711_WELD_BUFF_DATA5.RBT22_BT_CODE_NO := W#16#0;
   S711_WELD_BUFF_DATA5.RBT22_WELD_COUNT := W#16#0;
   S711_WELD_BUFF_DATA5.RBT23_BT_CODE_NO := W#16#0;
   S711_WELD_BUFF_DATA5.RBT23_WELD_COUNT := W#16#0;
   S711_WELD_BUFF_DATA5.RBT24_BT_CODE_NO := W#16#0;
   S711_WELD_BUFF_DATA5.RBT24_WELD_COUNT := W#16#0;
   S711_WELD_BUFF_DATA5.WELD_DETERMINES_RESULT := W#16#0;
   S711_WELD_BUFF_DATA5.WELD_CHECK_SUM := W#16#0;
   S711_WELD_BUFF_DATA5.SPARE1 := W#16#0;
   S711_WELD_BUFF_DATA6.STATION_MAIN := W#16#0;
   S711_WELD_BUFF_DATA6.DISTINCTION_LH_RH := W#16#0;
   S711_WELD_BUFF_DATA6.STAION_NUMBER := W#16#0;
   S711_WELD_BUFF_DATA6.VIN_NUMBER1 := W#16#0;
   S711_WELD_BUFF_DATA6.VIN_NUMBER2 := W#16#0;
   S711_WELD_BUFF_DATA6.VIN_NUMBER3 := W#16#0;
   S711_WELD_BUFF_DATA6.VIN_NUMBER4 := W#16#0;
   S711_WELD_BUFF_DATA6.SEQ_NUMBER1 := W#16#0;
   S711_WELD_BUFF_DATA6.SEQ_NUMBER2 := W#16#0;
   S711_WELD_BUFF_DATA6.RBT1_BT_CODE_NO := W#16#0;
   S711_WELD_BUFF_DATA6.RBT1_WELD_COUNT := W#16#0;
   S711_WELD_BUFF_DATA6.RBT2_BT_CODE_NO := W#16#0;
   S711_WELD_BUFF_DATA6.RBT2_WELD_COUNT := W#16#0;
   S711_WELD_BUFF_DATA6.RBT3_BT_CODE_NO := W#16#0;
   S711_WELD_BUFF_DATA6.RBT3_WELD_COUNT := W#16#0;
   S711_WELD_BUFF_DATA6.RBT4_BT_CODE_NO := W#16#0;
   S711_WELD_BUFF_DATA6.RBT4_WELD_COUNT := W#16#0;
   S711_WELD_BUFF_DATA6.RBT5_BT_CODE_NO := W#16#0;
   S711_WELD_BUFF_DATA6.RBT5_WELD_COUNT := W#16#0;
   S711_WELD_BUFF_DATA6.RBT6_BT_CODE_NO := W#16#0;
   S711_WELD_BUFF_DATA6.RBT6_WELD_COUNT := W#16#0;
   S711_WELD_BUFF_DATA6.RBT7_BT_CODE_NO := W#16#0;
   S711_WELD_BUFF_DATA6.RBT7_WELD_COUNT := W#16#0;
   S711_WELD_BUFF_DATA6.RBT8_BT_CODE_NO := W#16#0;
   S711_WELD_BUFF_DATA6.RBT8_WELD_COUNT := W#16#0;
   S711_WELD_BUFF_DATA6.RBT9_BT_CODE_NO := W#16#0;
   S711_WELD_BUFF_DATA6.RBT9_WELD_COUNT := W#16#0;
   S711_WELD_BUFF_DATA6.RBT10_BT_CODE_NO := W#16#0;
   S711_WELD_BUFF_DATA6.RBT10_WELD_COUNT := W#16#0;
   S711_WELD_BUFF_DATA6.RBT11_BT_CODE_NO := W#16#0;
   S711_WELD_BUFF_DATA6.RBT11_WELD_COUNT := W#16#0;
   S711_WELD_BUFF_DATA6.RBT12_BT_CODE_NO := W#16#0;
   S711_WELD_BUFF_DATA6.RBT12_WELD_COUNT := W#16#0;
   S711_WELD_BUFF_DATA6.RBT13_BT_CODE_NO := W#16#0;
   S711_WELD_BUFF_DATA6.RBT13_WELD_COUNT := W#16#0;
   S711_WELD_BUFF_DATA6.RBT14_BT_CODE_NO := W#16#0;
   S711_WELD_BUFF_DATA6.RBT14_WELD_COUNT := W#16#0;
   S711_WELD_BUFF_DATA6.RBT15_BT_CODE_NO := W#16#0;
   S711_WELD_BUFF_DATA6.RBT15_WELD_COUNT := W#16#0;
   S711_WELD_BUFF_DATA6.RBT16_BT_CODE_NO := W#16#0;
   S711_WELD_BUFF_DATA6.RBT16_WELD_COUNT := W#16#0;
   S711_WELD_BUFF_DATA6.RBT17_BT_CODE_NO := W#16#0;
   S711_WELD_BUFF_DATA6.RBT17_WELD_COUNT := W#16#0;
   S711_WELD_BUFF_DATA6.RBT18_BT_CODE_NO := W#16#0;
   S711_WELD_BUFF_DATA6.RBT18_WELD_COUNT := W#16#0;
   S711_WELD_BUFF_DATA6.RBT19_BT_CODE_NO := W#16#0;
   S711_WELD_BUFF_DATA6.RBT19_WELD_COUNT := W#16#0;
   S711_WELD_BUFF_DATA6.RBT20_BT_CODE_NO := W#16#0;
   S711_WELD_BUFF_DATA6.RBT20_WELD_COUNT := W#16#0;
   S711_WELD_BUFF_DATA6.RBT21_BT_CODE_NO := W#16#0;
   S711_WELD_BUFF_DATA6.RBT21_WELD_COUNT := W#16#0;
   S711_WELD_BUFF_DATA6.RBT22_BT_CODE_NO := W#16#0;
   S711_WELD_BUFF_DATA6.RBT22_WELD_COUNT := W#16#0;
   S711_WELD_BUFF_DATA6.RBT23_BT_CODE_NO := W#16#0;
   S711_WELD_BUFF_DATA6.RBT23_WELD_COUNT := W#16#0;
   S711_WELD_BUFF_DATA6.RBT24_BT_CODE_NO := W#16#0;
   S711_WELD_BUFF_DATA6.RBT24_WELD_COUNT := W#16#0;
   S711_WELD_BUFF_DATA6.WELD_DETERMINES_RESULT := W#16#0;
   S711_WELD_BUFF_DATA6.WELD_CHECK_SUM := W#16#0;
   S711_WELD_BUFF_DATA6.SPARE1 := W#16#0;
   S711_WELD_BUFF_DATA7.STATION_MAIN := W#16#0;
   S711_WELD_BUFF_DATA7.DISTINCTION_LH_RH := W#16#0;
   S711_WELD_BUFF_DATA7.STAION_NUMBER := W#16#0;
   S711_WELD_BUFF_DATA7.VIN_NUMBER1 := W#16#0;
   S711_WELD_BUFF_DATA7.VIN_NUMBER2 := W#16#0;
   S711_WELD_BUFF_DATA7.VIN_NUMBER3 := W#16#0;
   S711_WELD_BUFF_DATA7.VIN_NUMBER4 := W#16#0;
   S711_WELD_BUFF_DATA7.SEQ_NUMBER1 := W#16#0;
   S711_WELD_BUFF_DATA7.SEQ_NUMBER2 := W#16#0;
   S711_WELD_BUFF_DATA7.RBT1_BT_CODE_NO := W#16#0;
   S711_WELD_BUFF_DATA7.RBT1_WELD_COUNT := W#16#0;
   S711_WELD_BUFF_DATA7.RBT2_BT_CODE_NO := W#16#0;
   S711_WELD_BUFF_DATA7.RBT2_WELD_COUNT := W#16#0;
   S711_WELD_BUFF_DATA7.RBT3_BT_CODE_NO := W#16#0;
   S711_WELD_BUFF_DATA7.RBT3_WELD_COUNT := W#16#0;
   S711_WELD_BUFF_DATA7.RBT4_BT_CODE_NO := W#16#0;
   S711_WELD_BUFF_DATA7.RBT4_WELD_COUNT := W#16#0;
   S711_WELD_BUFF_DATA7.RBT5_BT_CODE_NO := W#16#0;
   S711_WELD_BUFF_DATA7.RBT5_WELD_COUNT := W#16#0;
   S711_WELD_BUFF_DATA7.RBT6_BT_CODE_NO := W#16#0;
   S711_WELD_BUFF_DATA7.RBT6_WELD_COUNT := W#16#0;
   S711_WELD_BUFF_DATA7.RBT7_BT_CODE_NO := W#16#0;
   S711_WELD_BUFF_DATA7.RBT7_WELD_COUNT := W#16#0;
   S711_WELD_BUFF_DATA7.RBT8_BT_CODE_NO := W#16#0;
   S711_WELD_BUFF_DATA7.RBT8_WELD_COUNT := W#16#0;
   S711_WELD_BUFF_DATA7.RBT9_BT_CODE_NO := W#16#0;
   S711_WELD_BUFF_DATA7.RBT9_WELD_COUNT := W#16#0;
   S711_WELD_BUFF_DATA7.RBT10_BT_CODE_NO := W#16#0;
   S711_WELD_BUFF_DATA7.RBT10_WELD_COUNT := W#16#0;
   S711_WELD_BUFF_DATA7.RBT11_BT_CODE_NO := W#16#0;
   S711_WELD_BUFF_DATA7.RBT11_WELD_COUNT := W#16#0;
   S711_WELD_BUFF_DATA7.RBT12_BT_CODE_NO := W#16#0;
   S711_WELD_BUFF_DATA7.RBT12_WELD_COUNT := W#16#0;
   S711_WELD_BUFF_DATA7.RBT13_BT_CODE_NO := W#16#0;
   S711_WELD_BUFF_DATA7.RBT13_WELD_COUNT := W#16#0;
   S711_WELD_BUFF_DATA7.RBT14_BT_CODE_NO := W#16#0;
   S711_WELD_BUFF_DATA7.RBT14_WELD_COUNT := W#16#0;
   S711_WELD_BUFF_DATA7.RBT15_BT_CODE_NO := W#16#0;
   S711_WELD_BUFF_DATA7.RBT15_WELD_COUNT := W#16#0;
   S711_WELD_BUFF_DATA7.RBT16_BT_CODE_NO := W#16#0;
   S711_WELD_BUFF_DATA7.RBT16_WELD_COUNT := W#16#0;
   S711_WELD_BUFF_DATA7.RBT17_BT_CODE_NO := W#16#0;
   S711_WELD_BUFF_DATA7.RBT17_WELD_COUNT := W#16#0;
   S711_WELD_BUFF_DATA7.RBT18_BT_CODE_NO := W#16#0;
   S711_WELD_BUFF_DATA7.RBT18_WELD_COUNT := W#16#0;
   S711_WELD_BUFF_DATA7.RBT19_BT_CODE_NO := W#16#0;
   S711_WELD_BUFF_DATA7.RBT19_WELD_COUNT := W#16#0;
   S711_WELD_BUFF_DATA7.RBT20_BT_CODE_NO := W#16#0;
   S711_WELD_BUFF_DATA7.RBT20_WELD_COUNT := W#16#0;
   S711_WELD_BUFF_DATA7.RBT21_BT_CODE_NO := W#16#0;
   S711_WELD_BUFF_DATA7.RBT21_WELD_COUNT := W#16#0;
   S711_WELD_BUFF_DATA7.RBT22_BT_CODE_NO := W#16#0;
   S711_WELD_BUFF_DATA7.RBT22_WELD_COUNT := W#16#0;
   S711_WELD_BUFF_DATA7.RBT23_BT_CODE_NO := W#16#0;
   S711_WELD_BUFF_DATA7.RBT23_WELD_COUNT := W#16#0;
   S711_WELD_BUFF_DATA7.RBT24_BT_CODE_NO := W#16#0;
   S711_WELD_BUFF_DATA7.RBT24_WELD_COUNT := W#16#0;
   S711_WELD_BUFF_DATA7.WELD_DETERMINES_RESULT := W#16#0;
   S711_WELD_BUFF_DATA7.WELD_CHECK_SUM := W#16#0;
   S711_WELD_BUFF_DATA7.SPARE1 := W#16#0;
   S711_WELD_BUFF_DATA8.STATION_MAIN := W#16#0;
   S711_WELD_BUFF_DATA8.DISTINCTION_LH_RH := W#16#0;
   S711_WELD_BUFF_DATA8.STAION_NUMBER := W#16#0;
   S711_WELD_BUFF_DATA8.VIN_NUMBER1 := W#16#0;
   S711_WELD_BUFF_DATA8.VIN_NUMBER2 := W#16#0;
   S711_WELD_BUFF_DATA8.VIN_NUMBER3 := W#16#0;
   S711_WELD_BUFF_DATA8.VIN_NUMBER4 := W#16#0;
   S711_WELD_BUFF_DATA8.SEQ_NUMBER1 := W#16#0;
   S711_WELD_BUFF_DATA8.SEQ_NUMBER2 := W#16#0;
   S711_WELD_BUFF_DATA8.RBT1_BT_CODE_NO := W#16#0;
   S711_WELD_BUFF_DATA8.RBT1_WELD_COUNT := W#16#0;
   S711_WELD_BUFF_DATA8.RBT2_BT_CODE_NO := W#16#0;
   S711_WELD_BUFF_DATA8.RBT2_WELD_COUNT := W#16#0;
   S711_WELD_BUFF_DATA8.RBT3_BT_CODE_NO := W#16#0;
   S711_WELD_BUFF_DATA8.RBT3_WELD_COUNT := W#16#0;
   S711_WELD_BUFF_DATA8.RBT4_BT_CODE_NO := W#16#0;
   S711_WELD_BUFF_DATA8.RBT4_WELD_COUNT := W#16#0;
   S711_WELD_BUFF_DATA8.RBT5_BT_CODE_NO := W#16#0;
   S711_WELD_BUFF_DATA8.RBT5_WELD_COUNT := W#16#0;
   S711_WELD_BUFF_DATA8.RBT6_BT_CODE_NO := W#16#0;
   S711_WELD_BUFF_DATA8.RBT6_WELD_COUNT := W#16#0;
   S711_WELD_BUFF_DATA8.RBT7_BT_CODE_NO := W#16#0;
   S711_WELD_BUFF_DATA8.RBT7_WELD_COUNT := W#16#0;
   S711_WELD_BUFF_DATA8.RBT8_BT_CODE_NO := W#16#0;
   S711_WELD_BUFF_DATA8.RBT8_WELD_COUNT := W#16#0;
   S711_WELD_BUFF_DATA8.RBT9_BT_CODE_NO := W#16#0;
   S711_WELD_BUFF_DATA8.RBT9_WELD_COUNT := W#16#0;
   S711_WELD_BUFF_DATA8.RBT10_BT_CODE_NO := W#16#0;
   S711_WELD_BUFF_DATA8.RBT10_WELD_COUNT := W#16#0;
   S711_WELD_BUFF_DATA8.RBT11_BT_CODE_NO := W#16#0;
   S711_WELD_BUFF_DATA8.RBT11_WELD_COUNT := W#16#0;
   S711_WELD_BUFF_DATA8.RBT12_BT_CODE_NO := W#16#0;
   S711_WELD_BUFF_DATA8.RBT12_WELD_COUNT := W#16#0;
   S711_WELD_BUFF_DATA8.RBT13_BT_CODE_NO := W#16#0;
   S711_WELD_BUFF_DATA8.RBT13_WELD_COUNT := W#16#0;
   S711_WELD_BUFF_DATA8.RBT14_BT_CODE_NO := W#16#0;
   S711_WELD_BUFF_DATA8.RBT14_WELD_COUNT := W#16#0;
   S711_WELD_BUFF_DATA8.RBT15_BT_CODE_NO := W#16#0;
   S711_WELD_BUFF_DATA8.RBT15_WELD_COUNT := W#16#0;
   S711_WELD_BUFF_DATA8.RBT16_BT_CODE_NO := W#16#0;
   S711_WELD_BUFF_DATA8.RBT16_WELD_COUNT := W#16#0;
   S711_WELD_BUFF_DATA8.RBT17_BT_CODE_NO := W#16#0;
   S711_WELD_BUFF_DATA8.RBT17_WELD_COUNT := W#16#0;
   S711_WELD_BUFF_DATA8.RBT18_BT_CODE_NO := W#16#0;
   S711_WELD_BUFF_DATA8.RBT18_WELD_COUNT := W#16#0;
   S711_WELD_BUFF_DATA8.RBT19_BT_CODE_NO := W#16#0;
   S711_WELD_BUFF_DATA8.RBT19_WELD_COUNT := W#16#0;
   S711_WELD_BUFF_DATA8.RBT20_BT_CODE_NO := W#16#0;
   S711_WELD_BUFF_DATA8.RBT20_WELD_COUNT := W#16#0;
   S711_WELD_BUFF_DATA8.RBT21_BT_CODE_NO := W#16#0;
   S711_WELD_BUFF_DATA8.RBT21_WELD_COUNT := W#16#0;
   S711_WELD_BUFF_DATA8.RBT22_BT_CODE_NO := W#16#0;
   S711_WELD_BUFF_DATA8.RBT22_WELD_COUNT := W#16#0;
   S711_WELD_BUFF_DATA8.RBT23_BT_CODE_NO := W#16#0;
   S711_WELD_BUFF_DATA8.RBT23_WELD_COUNT := W#16#0;
   S711_WELD_BUFF_DATA8.RBT24_BT_CODE_NO := W#16#0;
   S711_WELD_BUFF_DATA8.RBT24_WELD_COUNT := W#16#0;
   S711_WELD_BUFF_DATA8.WELD_DETERMINES_RESULT := W#16#0;
   S711_WELD_BUFF_DATA8.WELD_CHECK_SUM := W#16#0;
   S711_WELD_BUFF_DATA8.SPARE1 := W#16#0;
   S711_WELD_BUFF_DATA9.STATION_MAIN := W#16#0;
   S711_WELD_BUFF_DATA9.DISTINCTION_LH_RH := W#16#0;
   S711_WELD_BUFF_DATA9.STAION_NUMBER := W#16#0;
   S711_WELD_BUFF_DATA9.VIN_NUMBER1 := W#16#0;
   S711_WELD_BUFF_DATA9.VIN_NUMBER2 := W#16#0;
   S711_WELD_BUFF_DATA9.VIN_NUMBER3 := W#16#0;
   S711_WELD_BUFF_DATA9.VIN_NUMBER4 := W#16#0;
   S711_WELD_BUFF_DATA9.SEQ_NUMBER1 := W#16#0;
   S711_WELD_BUFF_DATA9.SEQ_NUMBER2 := W#16#0;
   S711_WELD_BUFF_DATA9.RBT1_BT_CODE_NO := W#16#0;
   S711_WELD_BUFF_DATA9.RBT1_WELD_COUNT := W#16#0;
   S711_WELD_BUFF_DATA9.RBT2_BT_CODE_NO := W#16#0;
   S711_WELD_BUFF_DATA9.RBT2_WELD_COUNT := W#16#0;
   S711_WELD_BUFF_DATA9.RBT3_BT_CODE_NO := W#16#0;
   S711_WELD_BUFF_DATA9.RBT3_WELD_COUNT := W#16#0;
   S711_WELD_BUFF_DATA9.RBT4_BT_CODE_NO := W#16#0;
   S711_WELD_BUFF_DATA9.RBT4_WELD_COUNT := W#16#0;
   S711_WELD_BUFF_DATA9.RBT5_BT_CODE_NO := W#16#0;
   S711_WELD_BUFF_DATA9.RBT5_WELD_COUNT := W#16#0;
   S711_WELD_BUFF_DATA9.RBT6_BT_CODE_NO := W#16#0;
   S711_WELD_BUFF_DATA9.RBT6_WELD_COUNT := W#16#0;
   S711_WELD_BUFF_DATA9.RBT7_BT_CODE_NO := W#16#0;
   S711_WELD_BUFF_DATA9.RBT7_WELD_COUNT := W#16#0;
   S711_WELD_BUFF_DATA9.RBT8_BT_CODE_NO := W#16#0;
   S711_WELD_BUFF_DATA9.RBT8_WELD_COUNT := W#16#0;
   S711_WELD_BUFF_DATA9.RBT9_BT_CODE_NO := W#16#0;
   S711_WELD_BUFF_DATA9.RBT9_WELD_COUNT := W#16#0;
   S711_WELD_BUFF_DATA9.RBT10_BT_CODE_NO := W#16#0;
   S711_WELD_BUFF_DATA9.RBT10_WELD_COUNT := W#16#0;
   S711_WELD_BUFF_DATA9.RBT11_BT_CODE_NO := W#16#0;
   S711_WELD_BUFF_DATA9.RBT11_WELD_COUNT := W#16#0;
   S711_WELD_BUFF_DATA9.RBT12_BT_CODE_NO := W#16#0;
   S711_WELD_BUFF_DATA9.RBT12_WELD_COUNT := W#16#0;
   S711_WELD_BUFF_DATA9.RBT13_BT_CODE_NO := W#16#0;
   S711_WELD_BUFF_DATA9.RBT13_WELD_COUNT := W#16#0;
   S711_WELD_BUFF_DATA9.RBT14_BT_CODE_NO := W#16#0;
   S711_WELD_BUFF_DATA9.RBT14_WELD_COUNT := W#16#0;
   S711_WELD_BUFF_DATA9.RBT15_BT_CODE_NO := W#16#0;
   S711_WELD_BUFF_DATA9.RBT15_WELD_COUNT := W#16#0;
   S711_WELD_BUFF_DATA9.RBT16_BT_CODE_NO := W#16#0;
   S711_WELD_BUFF_DATA9.RBT16_WELD_COUNT := W#16#0;
   S711_WELD_BUFF_DATA9.RBT17_BT_CODE_NO := W#16#0;
   S711_WELD_BUFF_DATA9.RBT17_WELD_COUNT := W#16#0;
   S711_WELD_BUFF_DATA9.RBT18_BT_CODE_NO := W#16#0;
   S711_WELD_BUFF_DATA9.RBT18_WELD_COUNT := W#16#0;
   S711_WELD_BUFF_DATA9.RBT19_BT_CODE_NO := W#16#0;
   S711_WELD_BUFF_DATA9.RBT19_WELD_COUNT := W#16#0;
   S711_WELD_BUFF_DATA9.RBT20_BT_CODE_NO := W#16#0;
   S711_WELD_BUFF_DATA9.RBT20_WELD_COUNT := W#16#0;
   S711_WELD_BUFF_DATA9.RBT21_BT_CODE_NO := W#16#0;
   S711_WELD_BUFF_DATA9.RBT21_WELD_COUNT := W#16#0;
   S711_WELD_BUFF_DATA9.RBT22_BT_CODE_NO := W#16#0;
   S711_WELD_BUFF_DATA9.RBT22_WELD_COUNT := W#16#0;
   S711_WELD_BUFF_DATA9.RBT23_BT_CODE_NO := W#16#0;
   S711_WELD_BUFF_DATA9.RBT23_WELD_COUNT := W#16#0;
   S711_WELD_BUFF_DATA9.RBT24_BT_CODE_NO := W#16#0;
   S711_WELD_BUFF_DATA9.RBT24_WELD_COUNT := W#16#0;
   S711_WELD_BUFF_DATA9.WELD_DETERMINES_RESULT := W#16#0;
   S711_WELD_BUFF_DATA9.WELD_CHECK_SUM := W#16#0;
   S711_WELD_BUFF_DATA9.SPARE1 := W#16#0;
   S711_WELD_BUFF_DATA10.STATION_MAIN := W#16#0;
   S711_WELD_BUFF_DATA10.DISTINCTION_LH_RH := W#16#0;
   S711_WELD_BUFF_DATA10.STAION_NUMBER := W#16#0;
   S711_WELD_BUFF_DATA10.VIN_NUMBER1 := W#16#0;
   S711_WELD_BUFF_DATA10.VIN_NUMBER2 := W#16#0;
   S711_WELD_BUFF_DATA10.VIN_NUMBER3 := W#16#0;
   S711_WELD_BUFF_DATA10.VIN_NUMBER4 := W#16#0;
   S711_WELD_BUFF_DATA10.SEQ_NUMBER1 := W#16#0;
   S711_WELD_BUFF_DATA10.SEQ_NUMBER2 := W#16#0;
   S711_WELD_BUFF_DATA10.RBT1_BT_CODE_NO := W#16#0;
   S711_WELD_BUFF_DATA10.RBT1_WELD_COUNT := W#16#0;
   S711_WELD_BUFF_DATA10.RBT2_BT_CODE_NO := W#16#0;
   S711_WELD_BUFF_DATA10.RBT2_WELD_COUNT := W#16#0;
   S711_WELD_BUFF_DATA10.RBT3_BT_CODE_NO := W#16#0;
   S711_WELD_BUFF_DATA10.RBT3_WELD_COUNT := W#16#0;
   S711_WELD_BUFF_DATA10.RBT4_BT_CODE_NO := W#16#0;
   S711_WELD_BUFF_DATA10.RBT4_WELD_COUNT := W#16#0;
   S711_WELD_BUFF_DATA10.RBT5_BT_CODE_NO := W#16#0;
   S711_WELD_BUFF_DATA10.RBT5_WELD_COUNT := W#16#0;
   S711_WELD_BUFF_DATA10.RBT6_BT_CODE_NO := W#16#0;
   S711_WELD_BUFF_DATA10.RBT6_WELD_COUNT := W#16#0;
   S711_WELD_BUFF_DATA10.RBT7_BT_CODE_NO := W#16#0;
   S711_WELD_BUFF_DATA10.RBT7_WELD_COUNT := W#16#0;
   S711_WELD_BUFF_DATA10.RBT8_BT_CODE_NO := W#16#0;
   S711_WELD_BUFF_DATA10.RBT8_WELD_COUNT := W#16#0;
   S711_WELD_BUFF_DATA10.RBT9_BT_CODE_NO := W#16#0;
   S711_WELD_BUFF_DATA10.RBT9_WELD_COUNT := W#16#0;
   S711_WELD_BUFF_DATA10.RBT10_BT_CODE_NO := W#16#0;
   S711_WELD_BUFF_DATA10.RBT10_WELD_COUNT := W#16#0;
   S711_WELD_BUFF_DATA10.RBT11_BT_CODE_NO := W#16#0;
   S711_WELD_BUFF_DATA10.RBT11_WELD_COUNT := W#16#0;
   S711_WELD_BUFF_DATA10.RBT12_BT_CODE_NO := W#16#0;
   S711_WELD_BUFF_DATA10.RBT12_WELD_COUNT := W#16#0;
   S711_WELD_BUFF_DATA10.RBT13_BT_CODE_NO := W#16#0;
   S711_WELD_BUFF_DATA10.RBT13_WELD_COUNT := W#16#0;
   S711_WELD_BUFF_DATA10.RBT14_BT_CODE_NO := W#16#0;
   S711_WELD_BUFF_DATA10.RBT14_WELD_COUNT := W#16#0;
   S711_WELD_BUFF_DATA10.RBT15_BT_CODE_NO := W#16#0;
   S711_WELD_BUFF_DATA10.RBT15_WELD_COUNT := W#16#0;
   S711_WELD_BUFF_DATA10.RBT16_BT_CODE_NO := W#16#0;
   S711_WELD_BUFF_DATA10.RBT16_WELD_COUNT := W#16#0;
   S711_WELD_BUFF_DATA10.RBT17_BT_CODE_NO := W#16#0;
   S711_WELD_BUFF_DATA10.RBT17_WELD_COUNT := W#16#0;
   S711_WELD_BUFF_DATA10.RBT18_BT_CODE_NO := W#16#0;
   S711_WELD_BUFF_DATA10.RBT18_WELD_COUNT := W#16#0;
   S711_WELD_BUFF_DATA10.RBT19_BT_CODE_NO := W#16#0;
   S711_WELD_BUFF_DATA10.RBT19_WELD_COUNT := W#16#0;
   S711_WELD_BUFF_DATA10.RBT20_BT_CODE_NO := W#16#0;
   S711_WELD_BUFF_DATA10.RBT20_WELD_COUNT := W#16#0;
   S711_WELD_BUFF_DATA10.RBT21_BT_CODE_NO := W#16#0;
   S711_WELD_BUFF_DATA10.RBT21_WELD_COUNT := W#16#0;
   S711_WELD_BUFF_DATA10.RBT22_BT_CODE_NO := W#16#0;
   S711_WELD_BUFF_DATA10.RBT22_WELD_COUNT := W#16#0;
   S711_WELD_BUFF_DATA10.RBT23_BT_CODE_NO := W#16#0;
   S711_WELD_BUFF_DATA10.RBT23_WELD_COUNT := W#16#0;
   S711_WELD_BUFF_DATA10.RBT24_BT_CODE_NO := W#16#0;
   S711_WELD_BUFF_DATA10.RBT24_WELD_COUNT := W#16#0;
   S711_WELD_BUFF_DATA10.WELD_DETERMINES_RESULT := W#16#0;
   S711_WELD_BUFF_DATA10.WELD_CHECK_SUM := W#16#0;
   S711_WELD_BUFF_DATA10.SPARE1 := W#16#0;
   S711_WELD_BUFF_DATA11.STATION_MAIN := W#16#0;
   S711_WELD_BUFF_DATA11.DISTINCTION_LH_RH := W#16#0;
   S711_WELD_BUFF_DATA11.STAION_NUMBER := W#16#0;
   S711_WELD_BUFF_DATA11.VIN_NUMBER1 := W#16#0;
   S711_WELD_BUFF_DATA11.VIN_NUMBER2 := W#16#0;
   S711_WELD_BUFF_DATA11.VIN_NUMBER3 := W#16#0;
   S711_WELD_BUFF_DATA11.VIN_NUMBER4 := W#16#0;
   S711_WELD_BUFF_DATA11.SEQ_NUMBER1 := W#16#0;
   S711_WELD_BUFF_DATA11.SEQ_NUMBER2 := W#16#0;
   S711_WELD_BUFF_DATA11.RBT1_BT_CODE_NO := W#16#0;
   S711_WELD_BUFF_DATA11.RBT1_WELD_COUNT := W#16#0;
   S711_WELD_BUFF_DATA11.RBT2_BT_CODE_NO := W#16#0;
   S711_WELD_BUFF_DATA11.RBT2_WELD_COUNT := W#16#0;
   S711_WELD_BUFF_DATA11.RBT3_BT_CODE_NO := W#16#0;
   S711_WELD_BUFF_DATA11.RBT3_WELD_COUNT := W#16#0;
   S711_WELD_BUFF_DATA11.RBT4_BT_CODE_NO := W#16#0;
   S711_WELD_BUFF_DATA11.RBT4_WELD_COUNT := W#16#0;
   S711_WELD_BUFF_DATA11.RBT5_BT_CODE_NO := W#16#0;
   S711_WELD_BUFF_DATA11.RBT5_WELD_COUNT := W#16#0;
   S711_WELD_BUFF_DATA11.RBT6_BT_CODE_NO := W#16#0;
   S711_WELD_BUFF_DATA11.RBT6_WELD_COUNT := W#16#0;
   S711_WELD_BUFF_DATA11.RBT7_BT_CODE_NO := W#16#0;
   S711_WELD_BUFF_DATA11.RBT7_WELD_COUNT := W#16#0;
   S711_WELD_BUFF_DATA11.RBT8_BT_CODE_NO := W#16#0;
   S711_WELD_BUFF_DATA11.RBT8_WELD_COUNT := W#16#0;
   S711_WELD_BUFF_DATA11.RBT9_BT_CODE_NO := W#16#0;
   S711_WELD_BUFF_DATA11.RBT9_WELD_COUNT := W#16#0;
   S711_WELD_BUFF_DATA11.RBT10_BT_CODE_NO := W#16#0;
   S711_WELD_BUFF_DATA11.RBT10_WELD_COUNT := W#16#0;
   S711_WELD_BUFF_DATA11.RBT11_BT_CODE_NO := W#16#0;
   S711_WELD_BUFF_DATA11.RBT11_WELD_COUNT := W#16#0;
   S711_WELD_BUFF_DATA11.RBT12_BT_CODE_NO := W#16#0;
   S711_WELD_BUFF_DATA11.RBT12_WELD_COUNT := W#16#0;
   S711_WELD_BUFF_DATA11.RBT13_BT_CODE_NO := W#16#0;
   S711_WELD_BUFF_DATA11.RBT13_WELD_COUNT := W#16#0;
   S711_WELD_BUFF_DATA11.RBT14_BT_CODE_NO := W#16#0;
   S711_WELD_BUFF_DATA11.RBT14_WELD_COUNT := W#16#0;
   S711_WELD_BUFF_DATA11.RBT15_BT_CODE_NO := W#16#0;
   S711_WELD_BUFF_DATA11.RBT15_WELD_COUNT := W#16#0;
   S711_WELD_BUFF_DATA11.RBT16_BT_CODE_NO := W#16#0;
   S711_WELD_BUFF_DATA11.RBT16_WELD_COUNT := W#16#0;
   S711_WELD_BUFF_DATA11.RBT17_BT_CODE_NO := W#16#0;
   S711_WELD_BUFF_DATA11.RBT17_WELD_COUNT := W#16#0;
   S711_WELD_BUFF_DATA11.RBT18_BT_CODE_NO := W#16#0;
   S711_WELD_BUFF_DATA11.RBT18_WELD_COUNT := W#16#0;
   S711_WELD_BUFF_DATA11.RBT19_BT_CODE_NO := W#16#0;
   S711_WELD_BUFF_DATA11.RBT19_WELD_COUNT := W#16#0;
   S711_WELD_BUFF_DATA11.RBT20_BT_CODE_NO := W#16#0;
   S711_WELD_BUFF_DATA11.RBT20_WELD_COUNT := W#16#0;
   S711_WELD_BUFF_DATA11.RBT21_BT_CODE_NO := W#16#0;
   S711_WELD_BUFF_DATA11.RBT21_WELD_COUNT := W#16#0;
   S711_WELD_BUFF_DATA11.RBT22_BT_CODE_NO := W#16#0;
   S711_WELD_BUFF_DATA11.RBT22_WELD_COUNT := W#16#0;
   S711_WELD_BUFF_DATA11.RBT23_BT_CODE_NO := W#16#0;
   S711_WELD_BUFF_DATA11.RBT23_WELD_COUNT := W#16#0;
   S711_WELD_BUFF_DATA11.RBT24_BT_CODE_NO := W#16#0;
   S711_WELD_BUFF_DATA11.RBT24_WELD_COUNT := W#16#0;
   S711_WELD_BUFF_DATA11.WELD_DETERMINES_RESULT := W#16#0;
   S711_WELD_BUFF_DATA11.WELD_CHECK_SUM := W#16#0;
   S711_WELD_BUFF_DATA11.SPARE1 := W#16#0;
   S711_WELD_BUFF_DATA21.STATION_MAIN := W#16#0;
   S711_WELD_BUFF_DATA21.DISTINCTION_LH_RH := W#16#0;
   S711_WELD_BUFF_DATA21.STAION_NUMBER := W#16#0;
   S711_WELD_BUFF_DATA21.VIN_NUMBER1 := W#16#0;
   S711_WELD_BUFF_DATA21.VIN_NUMBER2 := W#16#0;
   S711_WELD_BUFF_DATA21.VIN_NUMBER3 := W#16#0;
   S711_WELD_BUFF_DATA21.VIN_NUMBER4 := W#16#0;
   S711_WELD_BUFF_DATA21.SEQ_NUMBER1 := W#16#0;
   S711_WELD_BUFF_DATA21.SEQ_NUMBER2 := W#16#0;
   S711_WELD_BUFF_DATA21.RBT1_BT_CODE_NO := W#16#0;
   S711_WELD_BUFF_DATA21.RBT1_WELD_COUNT := W#16#0;
   S711_WELD_BUFF_DATA21.RBT2_BT_CODE_NO := W#16#0;
   S711_WELD_BUFF_DATA21.RBT2_WELD_COUNT := W#16#0;
   S711_WELD_BUFF_DATA21.RBT3_BT_CODE_NO := W#16#0;
   S711_WELD_BUFF_DATA21.RBT3_WELD_COUNT := W#16#0;
   S711_WELD_BUFF_DATA21.RBT4_BT_CODE_NO := W#16#0;
   S711_WELD_BUFF_DATA21.RBT4_WELD_COUNT := W#16#0;
   S711_WELD_BUFF_DATA21.RBT5_BT_CODE_NO := W#16#0;
   S711_WELD_BUFF_DATA21.RBT5_WELD_COUNT := W#16#0;
   S711_WELD_BUFF_DATA21.RBT6_BT_CODE_NO := W#16#0;
   S711_WELD_BUFF_DATA21.RBT6_WELD_COUNT := W#16#0;
   S711_WELD_BUFF_DATA21.RBT7_BT_CODE_NO := W#16#0;
   S711_WELD_BUFF_DATA21.RBT7_WELD_COUNT := W#16#0;
   S711_WELD_BUFF_DATA21.RBT8_BT_CODE_NO := W#16#0;
   S711_WELD_BUFF_DATA21.RBT8_WELD_COUNT := W#16#0;
   S711_WELD_BUFF_DATA21.RBT9_BT_CODE_NO := W#16#0;
   S711_WELD_BUFF_DATA21.RBT9_WELD_COUNT := W#16#0;
   S711_WELD_BUFF_DATA21.RBT10_BT_CODE_NO := W#16#0;
   S711_WELD_BUFF_DATA21.RBT10_WELD_COUNT := W#16#0;
   S711_WELD_BUFF_DATA21.RBT11_BT_CODE_NO := W#16#0;
   S711_WELD_BUFF_DATA21.RBT11_WELD_COUNT := W#16#0;
   S711_WELD_BUFF_DATA21.RBT12_BT_CODE_NO := W#16#0;
   S711_WELD_BUFF_DATA21.RBT12_WELD_COUNT := W#16#0;
   S711_WELD_BUFF_DATA21.RBT13_BT_CODE_NO := W#16#0;
   S711_WELD_BUFF_DATA21.RBT13_WELD_COUNT := W#16#0;
   S711_WELD_BUFF_DATA21.RBT14_BT_CODE_NO := W#16#0;
   S711_WELD_BUFF_DATA21.RBT14_WELD_COUNT := W#16#0;
   S711_WELD_BUFF_DATA21.RBT15_BT_CODE_NO := W#16#0;
   S711_WELD_BUFF_DATA21.RBT15_WELD_COUNT := W#16#0;
   S711_WELD_BUFF_DATA21.RBT16_BT_CODE_NO := W#16#0;
   S711_WELD_BUFF_DATA21.RBT16_WELD_COUNT := W#16#0;
   S711_WELD_BUFF_DATA21.RBT17_BT_CODE_NO := W#16#0;
   S711_WELD_BUFF_DATA21.RBT17_WELD_COUNT := W#16#0;
   S711_WELD_BUFF_DATA21.RBT18_BT_CODE_NO := W#16#0;
   S711_WELD_BUFF_DATA21.RBT18_WELD_COUNT := W#16#0;
   S711_WELD_BUFF_DATA21.RBT19_BT_CODE_NO := W#16#0;
   S711_WELD_BUFF_DATA21.RBT19_WELD_COUNT := W#16#0;
   S711_WELD_BUFF_DATA21.RBT20_BT_CODE_NO := W#16#0;
   S711_WELD_BUFF_DATA21.RBT20_WELD_COUNT := W#16#0;
   S711_WELD_BUFF_DATA21.RBT21_BT_CODE_NO := W#16#0;
   S711_WELD_BUFF_DATA21.RBT21_WELD_COUNT := W#16#0;
   S711_WELD_BUFF_DATA21.RBT22_BT_CODE_NO := W#16#0;
   S711_WELD_BUFF_DATA21.RBT22_WELD_COUNT := W#16#0;
   S711_WELD_BUFF_DATA21.RBT23_BT_CODE_NO := W#16#0;
   S711_WELD_BUFF_DATA21.RBT23_WELD_COUNT := W#16#0;
   S711_WELD_BUFF_DATA21.RBT24_BT_CODE_NO := W#16#0;
   S711_WELD_BUFF_DATA21.RBT24_WELD_COUNT := W#16#0;
   S711_WELD_BUFF_DATA21.WELD_DETERMINES_RESULT := W#16#0;
   S711_WELD_BUFF_DATA21.WELD_CHECK_SUM := W#16#0;
   S711_WELD_BUFF_DATA21.SPARE1 := W#16#0;
   S711_WELD_BUFF_DATA31.STATION_MAIN := W#16#0;
   S711_WELD_BUFF_DATA31.DISTINCTION_LH_RH := W#16#0;
   S711_WELD_BUFF_DATA31.STAION_NUMBER := W#16#0;
   S711_WELD_BUFF_DATA31.VIN_NUMBER1 := W#16#0;
   S711_WELD_BUFF_DATA31.VIN_NUMBER2 := W#16#0;
   S711_WELD_BUFF_DATA31.VIN_NUMBER3 := W#16#0;
   S711_WELD_BUFF_DATA31.VIN_NUMBER4 := W#16#0;
   S711_WELD_BUFF_DATA31.SEQ_NUMBER1 := W#16#0;
   S711_WELD_BUFF_DATA31.SEQ_NUMBER2 := W#16#0;
   S711_WELD_BUFF_DATA31.RBT1_BT_CODE_NO := W#16#0;
   S711_WELD_BUFF_DATA31.RBT1_WELD_COUNT := W#16#0;
   S711_WELD_BUFF_DATA31.RBT2_BT_CODE_NO := W#16#0;
   S711_WELD_BUFF_DATA31.RBT2_WELD_COUNT := W#16#0;
   S711_WELD_BUFF_DATA31.RBT3_BT_CODE_NO := W#16#0;
   S711_WELD_BUFF_DATA31.RBT3_WELD_COUNT := W#16#0;
   S711_WELD_BUFF_DATA31.RBT4_BT_CODE_NO := W#16#0;
   S711_WELD_BUFF_DATA31.RBT4_WELD_COUNT := W#16#0;
   S711_WELD_BUFF_DATA31.RBT5_BT_CODE_NO := W#16#0;
   S711_WELD_BUFF_DATA31.RBT5_WELD_COUNT := W#16#0;
   S711_WELD_BUFF_DATA31.RBT6_BT_CODE_NO := W#16#0;
   S711_WELD_BUFF_DATA31.RBT6_WELD_COUNT := W#16#0;
   S711_WELD_BUFF_DATA31.RBT7_BT_CODE_NO := W#16#0;
   S711_WELD_BUFF_DATA31.RBT7_WELD_COUNT := W#16#0;
   S711_WELD_BUFF_DATA31.RBT8_BT_CODE_NO := W#16#0;
   S711_WELD_BUFF_DATA31.RBT8_WELD_COUNT := W#16#0;
   S711_WELD_BUFF_DATA31.RBT9_BT_CODE_NO := W#16#0;
   S711_WELD_BUFF_DATA31.RBT9_WELD_COUNT := W#16#0;
   S711_WELD_BUFF_DATA31.RBT10_BT_CODE_NO := W#16#0;
   S711_WELD_BUFF_DATA31.RBT10_WELD_COUNT := W#16#0;
   S711_WELD_BUFF_DATA31.RBT11_BT_CODE_NO := W#16#0;
   S711_WELD_BUFF_DATA31.RBT11_WELD_COUNT := W#16#0;
   S711_WELD_BUFF_DATA31.RBT12_BT_CODE_NO := W#16#0;
   S711_WELD_BUFF_DATA31.RBT12_WELD_COUNT := W#16#0;
   S711_WELD_BUFF_DATA31.RBT13_BT_CODE_NO := W#16#0;
   S711_WELD_BUFF_DATA31.RBT13_WELD_COUNT := W#16#0;
   S711_WELD_BUFF_DATA31.RBT14_BT_CODE_NO := W#16#0;
   S711_WELD_BUFF_DATA31.RBT14_WELD_COUNT := W#16#0;
   S711_WELD_BUFF_DATA31.RBT15_BT_CODE_NO := W#16#0;
   S711_WELD_BUFF_DATA31.RBT15_WELD_COUNT := W#16#0;
   S711_WELD_BUFF_DATA31.RBT16_BT_CODE_NO := W#16#0;
   S711_WELD_BUFF_DATA31.RBT16_WELD_COUNT := W#16#0;
   S711_WELD_BUFF_DATA31.RBT17_BT_CODE_NO := W#16#0;
   S711_WELD_BUFF_DATA31.RBT17_WELD_COUNT := W#16#0;
   S711_WELD_BUFF_DATA31.RBT18_BT_CODE_NO := W#16#0;
   S711_WELD_BUFF_DATA31.RBT18_WELD_COUNT := W#16#0;
   S711_WELD_BUFF_DATA31.RBT19_BT_CODE_NO := W#16#0;
   S711_WELD_BUFF_DATA31.RBT19_WELD_COUNT := W#16#0;
   S711_WELD_BUFF_DATA31.RBT20_BT_CODE_NO := W#16#0;
   S711_WELD_BUFF_DATA31.RBT20_WELD_COUNT := W#16#0;
   S711_WELD_BUFF_DATA31.RBT21_BT_CODE_NO := W#16#0;
   S711_WELD_BUFF_DATA31.RBT21_WELD_COUNT := W#16#0;
   S711_WELD_BUFF_DATA31.RBT22_BT_CODE_NO := W#16#0;
   S711_WELD_BUFF_DATA31.RBT22_WELD_COUNT := W#16#0;
   S711_WELD_BUFF_DATA31.RBT23_BT_CODE_NO := W#16#0;
   S711_WELD_BUFF_DATA31.RBT23_WELD_COUNT := W#16#0;
   S711_WELD_BUFF_DATA31.RBT24_BT_CODE_NO := W#16#0;
   S711_WELD_BUFF_DATA31.RBT24_WELD_COUNT := W#16#0;
   S711_WELD_BUFF_DATA31.WELD_DETERMINES_RESULT := W#16#0;
   S711_WELD_BUFF_DATA31.WELD_CHECK_SUM := W#16#0;
   S711_WELD_BUFF_DATA31.SPARE1 := W#16#0;
   S711_WELD_BUFF_DATA41.STATION_MAIN := W#16#0;
   S711_WELD_BUFF_DATA41.DISTINCTION_LH_RH := W#16#0;
   S711_WELD_BUFF_DATA41.STAION_NUMBER := W#16#0;
   S711_WELD_BUFF_DATA41.VIN_NUMBER1 := W#16#0;
   S711_WELD_BUFF_DATA41.VIN_NUMBER2 := W#16#0;
   S711_WELD_BUFF_DATA41.VIN_NUMBER3 := W#16#0;
   S711_WELD_BUFF_DATA41.VIN_NUMBER4 := W#16#0;
   S711_WELD_BUFF_DATA41.SEQ_NUMBER1 := W#16#0;
   S711_WELD_BUFF_DATA41.SEQ_NUMBER2 := W#16#0;
   S711_WELD_BUFF_DATA41.RBT1_BT_CODE_NO := W#16#0;
   S711_WELD_BUFF_DATA41.RBT1_WELD_COUNT := W#16#0;
   S711_WELD_BUFF_DATA41.RBT2_BT_CODE_NO := W#16#0;
   S711_WELD_BUFF_DATA41.RBT2_WELD_COUNT := W#16#0;
   S711_WELD_BUFF_DATA41.RBT3_BT_CODE_NO := W#16#0;
   S711_WELD_BUFF_DATA41.RBT3_WELD_COUNT := W#16#0;
   S711_WELD_BUFF_DATA41.RBT4_BT_CODE_NO := W#16#0;
   S711_WELD_BUFF_DATA41.RBT4_WELD_COUNT := W#16#0;
   S711_WELD_BUFF_DATA41.RBT5_BT_CODE_NO := W#16#0;
   S711_WELD_BUFF_DATA41.RBT5_WELD_COUNT := W#16#0;
   S711_WELD_BUFF_DATA41.RBT6_BT_CODE_NO := W#16#0;
   S711_WELD_BUFF_DATA41.RBT6_WELD_COUNT := W#16#0;
   S711_WELD_BUFF_DATA41.RBT7_BT_CODE_NO := W#16#0;
   S711_WELD_BUFF_DATA41.RBT7_WELD_COUNT := W#16#0;
   S711_WELD_BUFF_DATA41.RBT8_BT_CODE_NO := W#16#0;
   S711_WELD_BUFF_DATA41.RBT8_WELD_COUNT := W#16#0;
   S711_WELD_BUFF_DATA41.RBT9_BT_CODE_NO := W#16#0;
   S711_WELD_BUFF_DATA41.RBT9_WELD_COUNT := W#16#0;
   S711_WELD_BUFF_DATA41.RBT10_BT_CODE_NO := W#16#0;
   S711_WELD_BUFF_DATA41.RBT10_WELD_COUNT := W#16#0;
   S711_WELD_BUFF_DATA41.RBT11_BT_CODE_NO := W#16#0;
   S711_WELD_BUFF_DATA41.RBT11_WELD_COUNT := W#16#0;
   S711_WELD_BUFF_DATA41.RBT12_BT_CODE_NO := W#16#0;
   S711_WELD_BUFF_DATA41.RBT12_WELD_COUNT := W#16#0;
   S711_WELD_BUFF_DATA41.RBT13_BT_CODE_NO := W#16#0;
   S711_WELD_BUFF_DATA41.RBT13_WELD_COUNT := W#16#0;
   S711_WELD_BUFF_DATA41.RBT14_BT_CODE_NO := W#16#0;
   S711_WELD_BUFF_DATA41.RBT14_WELD_COUNT := W#16#0;
   S711_WELD_BUFF_DATA41.RBT15_BT_CODE_NO := W#16#0;
   S711_WELD_BUFF_DATA41.RBT15_WELD_COUNT := W#16#0;
   S711_WELD_BUFF_DATA41.RBT16_BT_CODE_NO := W#16#0;
   S711_WELD_BUFF_DATA41.RBT16_WELD_COUNT := W#16#0;
   S711_WELD_BUFF_DATA41.RBT17_BT_CODE_NO := W#16#0;
   S711_WELD_BUFF_DATA41.RBT17_WELD_COUNT := W#16#0;
   S711_WELD_BUFF_DATA41.RBT18_BT_CODE_NO := W#16#0;
   S711_WELD_BUFF_DATA41.RBT18_WELD_COUNT := W#16#0;
   S711_WELD_BUFF_DATA41.RBT19_BT_CODE_NO := W#16#0;
   S711_WELD_BUFF_DATA41.RBT19_WELD_COUNT := W#16#0;
   S711_WELD_BUFF_DATA41.RBT20_BT_CODE_NO := W#16#0;
   S711_WELD_BUFF_DATA41.RBT20_WELD_COUNT := W#16#0;
   S711_WELD_BUFF_DATA41.RBT21_BT_CODE_NO := W#16#0;
   S711_WELD_BUFF_DATA41.RBT21_WELD_COUNT := W#16#0;
   S711_WELD_BUFF_DATA41.RBT22_BT_CODE_NO := W#16#0;
   S711_WELD_BUFF_DATA41.RBT22_WELD_COUNT := W#16#0;
   S711_WELD_BUFF_DATA41.RBT23_BT_CODE_NO := W#16#0;
   S711_WELD_BUFF_DATA41.RBT23_WELD_COUNT := W#16#0;
   S711_WELD_BUFF_DATA41.RBT24_BT_CODE_NO := W#16#0;
   S711_WELD_BUFF_DATA41.RBT24_WELD_COUNT := W#16#0;
   S711_WELD_BUFF_DATA41.WELD_DETERMINES_RESULT := W#16#0;
   S711_WELD_BUFF_DATA41.WELD_CHECK_SUM := W#16#0;
   S711_WELD_BUFF_DATA41.SPARE1 := W#16#0;
   S711_WELD_BUFF_DATA51.STATION_MAIN := W#16#0;
   S711_WELD_BUFF_DATA51.DISTINCTION_LH_RH := W#16#0;
   S711_WELD_BUFF_DATA51.STAION_NUMBER := W#16#0;
   S711_WELD_BUFF_DATA51.VIN_NUMBER1 := W#16#0;
   S711_WELD_BUFF_DATA51.VIN_NUMBER2 := W#16#0;
   S711_WELD_BUFF_DATA51.VIN_NUMBER3 := W#16#0;
   S711_WELD_BUFF_DATA51.VIN_NUMBER4 := W#16#0;
   S711_WELD_BUFF_DATA51.SEQ_NUMBER1 := W#16#0;
   S711_WELD_BUFF_DATA51.SEQ_NUMBER2 := W#16#0;
   S711_WELD_BUFF_DATA51.RBT1_BT_CODE_NO := W#16#0;
   S711_WELD_BUFF_DATA51.RBT1_WELD_COUNT := W#16#0;
   S711_WELD_BUFF_DATA51.RBT2_BT_CODE_NO := W#16#0;
   S711_WELD_BUFF_DATA51.RBT2_WELD_COUNT := W#16#0;
   S711_WELD_BUFF_DATA51.RBT3_BT_CODE_NO := W#16#0;
   S711_WELD_BUFF_DATA51.RBT3_WELD_COUNT := W#16#0;
   S711_WELD_BUFF_DATA51.RBT4_BT_CODE_NO := W#16#0;
   S711_WELD_BUFF_DATA51.RBT4_WELD_COUNT := W#16#0;
   S711_WELD_BUFF_DATA51.RBT5_BT_CODE_NO := W#16#0;
   S711_WELD_BUFF_DATA51.RBT5_WELD_COUNT := W#16#0;
   S711_WELD_BUFF_DATA51.RBT6_BT_CODE_NO := W#16#0;
   S711_WELD_BUFF_DATA51.RBT6_WELD_COUNT := W#16#0;
   S711_WELD_BUFF_DATA51.RBT7_BT_CODE_NO := W#16#0;
   S711_WELD_BUFF_DATA51.RBT7_WELD_COUNT := W#16#0;
   S711_WELD_BUFF_DATA51.RBT8_BT_CODE_NO := W#16#0;
   S711_WELD_BUFF_DATA51.RBT8_WELD_COUNT := W#16#0;
   S711_WELD_BUFF_DATA51.RBT9_BT_CODE_NO := W#16#0;
   S711_WELD_BUFF_DATA51.RBT9_WELD_COUNT := W#16#0;
   S711_WELD_BUFF_DATA51.RBT10_BT_CODE_NO := W#16#0;
   S711_WELD_BUFF_DATA51.RBT10_WELD_COUNT := W#16#0;
   S711_WELD_BUFF_DATA51.RBT11_BT_CODE_NO := W#16#0;
   S711_WELD_BUFF_DATA51.RBT11_WELD_COUNT := W#16#0;
   S711_WELD_BUFF_DATA51.RBT12_BT_CODE_NO := W#16#0;
   S711_WELD_BUFF_DATA51.RBT12_WELD_COUNT := W#16#0;
   S711_WELD_BUFF_DATA51.RBT13_BT_CODE_NO := W#16#0;
   S711_WELD_BUFF_DATA51.RBT13_WELD_COUNT := W#16#0;
   S711_WELD_BUFF_DATA51.RBT14_BT_CODE_NO := W#16#0;
   S711_WELD_BUFF_DATA51.RBT14_WELD_COUNT := W#16#0;
   S711_WELD_BUFF_DATA51.RBT15_BT_CODE_NO := W#16#0;
   S711_WELD_BUFF_DATA51.RBT15_WELD_COUNT := W#16#0;
   S711_WELD_BUFF_DATA51.RBT16_BT_CODE_NO := W#16#0;
   S711_WELD_BUFF_DATA51.RBT16_WELD_COUNT := W#16#0;
   S711_WELD_BUFF_DATA51.RBT17_BT_CODE_NO := W#16#0;
   S711_WELD_BUFF_DATA51.RBT17_WELD_COUNT := W#16#0;
   S711_WELD_BUFF_DATA51.RBT18_BT_CODE_NO := W#16#0;
   S711_WELD_BUFF_DATA51.RBT18_WELD_COUNT := W#16#0;
   S711_WELD_BUFF_DATA51.RBT19_BT_CODE_NO := W#16#0;
   S711_WELD_BUFF_DATA51.RBT19_WELD_COUNT := W#16#0;
   S711_WELD_BUFF_DATA51.RBT20_BT_CODE_NO := W#16#0;
   S711_WELD_BUFF_DATA51.RBT20_WELD_COUNT := W#16#0;
   S711_WELD_BUFF_DATA51.RBT21_BT_CODE_NO := W#16#0;
   S711_WELD_BUFF_DATA51.RBT21_WELD_COUNT := W#16#0;
   S711_WELD_BUFF_DATA51.RBT22_BT_CODE_NO := W#16#0;
   S711_WELD_BUFF_DATA51.RBT22_WELD_COUNT := W#16#0;
   S711_WELD_BUFF_DATA51.RBT23_BT_CODE_NO := W#16#0;
   S711_WELD_BUFF_DATA51.RBT23_WELD_COUNT := W#16#0;
   S711_WELD_BUFF_DATA51.RBT24_BT_CODE_NO := W#16#0;
   S711_WELD_BUFF_DATA51.RBT24_WELD_COUNT := W#16#0;
   S711_WELD_BUFF_DATA51.WELD_DETERMINES_RESULT := W#16#0;
   S711_WELD_BUFF_DATA51.WELD_CHECK_SUM := W#16#0;
   S711_WELD_BUFF_DATA51.SPARE1 := W#16#0;
   S711_WELD_BUFF_DATA61.STATION_MAIN := W#16#0;
   S711_WELD_BUFF_DATA61.DISTINCTION_LH_RH := W#16#0;
   S711_WELD_BUFF_DATA61.STAION_NUMBER := W#16#0;
   S711_WELD_BUFF_DATA61.VIN_NUMBER1 := W#16#0;
   S711_WELD_BUFF_DATA61.VIN_NUMBER2 := W#16#0;
   S711_WELD_BUFF_DATA61.VIN_NUMBER3 := W#16#0;
   S711_WELD_BUFF_DATA61.VIN_NUMBER4 := W#16#0;
   S711_WELD_BUFF_DATA61.SEQ_NUMBER1 := W#16#0;
   S711_WELD_BUFF_DATA61.SEQ_NUMBER2 := W#16#0;
   S711_WELD_BUFF_DATA61.RBT1_BT_CODE_NO := W#16#0;
   S711_WELD_BUFF_DATA61.RBT1_WELD_COUNT := W#16#0;
   S711_WELD_BUFF_DATA61.RBT2_BT_CODE_NO := W#16#0;
   S711_WELD_BUFF_DATA61.RBT2_WELD_COUNT := W#16#0;
   S711_WELD_BUFF_DATA61.RBT3_BT_CODE_NO := W#16#0;
   S711_WELD_BUFF_DATA61.RBT3_WELD_COUNT := W#16#0;
   S711_WELD_BUFF_DATA61.RBT4_BT_CODE_NO := W#16#0;
   S711_WELD_BUFF_DATA61.RBT4_WELD_COUNT := W#16#0;
   S711_WELD_BUFF_DATA61.RBT5_BT_CODE_NO := W#16#0;
   S711_WELD_BUFF_DATA61.RBT5_WELD_COUNT := W#16#0;
   S711_WELD_BUFF_DATA61.RBT6_BT_CODE_NO := W#16#0;
   S711_WELD_BUFF_DATA61.RBT6_WELD_COUNT := W#16#0;
   S711_WELD_BUFF_DATA61.RBT7_BT_CODE_NO := W#16#0;
   S711_WELD_BUFF_DATA61.RBT7_WELD_COUNT := W#16#0;
   S711_WELD_BUFF_DATA61.RBT8_BT_CODE_NO := W#16#0;
   S711_WELD_BUFF_DATA61.RBT8_WELD_COUNT := W#16#0;
   S711_WELD_BUFF_DATA61.RBT9_BT_CODE_NO := W#16#0;
   S711_WELD_BUFF_DATA61.RBT9_WELD_COUNT := W#16#0;
   S711_WELD_BUFF_DATA61.RBT10_BT_CODE_NO := W#16#0;
   S711_WELD_BUFF_DATA61.RBT10_WELD_COUNT := W#16#0;
   S711_WELD_BUFF_DATA61.RBT11_BT_CODE_NO := W#16#0;
   S711_WELD_BUFF_DATA61.RBT11_WELD_COUNT := W#16#0;
   S711_WELD_BUFF_DATA61.RBT12_BT_CODE_NO := W#16#0;
   S711_WELD_BUFF_DATA61.RBT12_WELD_COUNT := W#16#0;
   S711_WELD_BUFF_DATA61.RBT13_BT_CODE_NO := W#16#0;
   S711_WELD_BUFF_DATA61.RBT13_WELD_COUNT := W#16#0;
   S711_WELD_BUFF_DATA61.RBT14_BT_CODE_NO := W#16#0;
   S711_WELD_BUFF_DATA61.RBT14_WELD_COUNT := W#16#0;
   S711_WELD_BUFF_DATA61.RBT15_BT_CODE_NO := W#16#0;
   S711_WELD_BUFF_DATA61.RBT15_WELD_COUNT := W#16#0;
   S711_WELD_BUFF_DATA61.RBT16_BT_CODE_NO := W#16#0;
   S711_WELD_BUFF_DATA61.RBT16_WELD_COUNT := W#16#0;
   S711_WELD_BUFF_DATA61.RBT17_BT_CODE_NO := W#16#0;
   S711_WELD_BUFF_DATA61.RBT17_WELD_COUNT := W#16#0;
   S711_WELD_BUFF_DATA61.RBT18_BT_CODE_NO := W#16#0;
   S711_WELD_BUFF_DATA61.RBT18_WELD_COUNT := W#16#0;
   S711_WELD_BUFF_DATA61.RBT19_BT_CODE_NO := W#16#0;
   S711_WELD_BUFF_DATA61.RBT19_WELD_COUNT := W#16#0;
   S711_WELD_BUFF_DATA61.RBT20_BT_CODE_NO := W#16#0;
   S711_WELD_BUFF_DATA61.RBT20_WELD_COUNT := W#16#0;
   S711_WELD_BUFF_DATA61.RBT21_BT_CODE_NO := W#16#0;
   S711_WELD_BUFF_DATA61.RBT21_WELD_COUNT := W#16#0;
   S711_WELD_BUFF_DATA61.RBT22_BT_CODE_NO := W#16#0;
   S711_WELD_BUFF_DATA61.RBT22_WELD_COUNT := W#16#0;
   S711_WELD_BUFF_DATA61.RBT23_BT_CODE_NO := W#16#0;
   S711_WELD_BUFF_DATA61.RBT23_WELD_COUNT := W#16#0;
   S711_WELD_BUFF_DATA61.RBT24_BT_CODE_NO := W#16#0;
   S711_WELD_BUFF_DATA61.RBT24_WELD_COUNT := W#16#0;
   S711_WELD_BUFF_DATA61.WELD_DETERMINES_RESULT := W#16#0;
   S711_WELD_BUFF_DATA61.WELD_CHECK_SUM := W#16#0;
   S711_WELD_BUFF_DATA61.SPARE1 := W#16#0;
   S711_WELD_BUFF_DATA71.STATION_MAIN := W#16#0;
   S711_WELD_BUFF_DATA71.DISTINCTION_LH_RH := W#16#0;
   S711_WELD_BUFF_DATA71.STAION_NUMBER := W#16#0;
   S711_WELD_BUFF_DATA71.VIN_NUMBER1 := W#16#0;
   S711_WELD_BUFF_DATA71.VIN_NUMBER2 := W#16#0;
   S711_WELD_BUFF_DATA71.VIN_NUMBER3 := W#16#0;
   S711_WELD_BUFF_DATA71.VIN_NUMBER4 := W#16#0;
   S711_WELD_BUFF_DATA71.SEQ_NUMBER1 := W#16#0;
   S711_WELD_BUFF_DATA71.SEQ_NUMBER2 := W#16#0;
   S711_WELD_BUFF_DATA71.RBT1_BT_CODE_NO := W#16#0;
   S711_WELD_BUFF_DATA71.RBT1_WELD_COUNT := W#16#0;
   S711_WELD_BUFF_DATA71.RBT2_BT_CODE_NO := W#16#0;
   S711_WELD_BUFF_DATA71.RBT2_WELD_COUNT := W#16#0;
   S711_WELD_BUFF_DATA71.RBT3_BT_CODE_NO := W#16#0;
   S711_WELD_BUFF_DATA71.RBT3_WELD_COUNT := W#16#0;
   S711_WELD_BUFF_DATA71.RBT4_BT_CODE_NO := W#16#0;
   S711_WELD_BUFF_DATA71.RBT4_WELD_COUNT := W#16#0;
   S711_WELD_BUFF_DATA71.RBT5_BT_CODE_NO := W#16#0;
   S711_WELD_BUFF_DATA71.RBT5_WELD_COUNT := W#16#0;
   S711_WELD_BUFF_DATA71.RBT6_BT_CODE_NO := W#16#0;
   S711_WELD_BUFF_DATA71.RBT6_WELD_COUNT := W#16#0;
   S711_WELD_BUFF_DATA71.RBT7_BT_CODE_NO := W#16#0;
   S711_WELD_BUFF_DATA71.RBT7_WELD_COUNT := W#16#0;
   S711_WELD_BUFF_DATA71.RBT8_BT_CODE_NO := W#16#0;
   S711_WELD_BUFF_DATA71.RBT8_WELD_COUNT := W#16#0;
   S711_WELD_BUFF_DATA71.RBT9_BT_CODE_NO := W#16#0;
   S711_WELD_BUFF_DATA71.RBT9_WELD_COUNT := W#16#0;
   S711_WELD_BUFF_DATA71.RBT10_BT_CODE_NO := W#16#0;
   S711_WELD_BUFF_DATA71.RBT10_WELD_COUNT := W#16#0;
   S711_WELD_BUFF_DATA71.RBT11_BT_CODE_NO := W#16#0;
   S711_WELD_BUFF_DATA71.RBT11_WELD_COUNT := W#16#0;
   S711_WELD_BUFF_DATA71.RBT12_BT_CODE_NO := W#16#0;
   S711_WELD_BUFF_DATA71.RBT12_WELD_COUNT := W#16#0;
   S711_WELD_BUFF_DATA71.RBT13_BT_CODE_NO := W#16#0;
   S711_WELD_BUFF_DATA71.RBT13_WELD_COUNT := W#16#0;
   S711_WELD_BUFF_DATA71.RBT14_BT_CODE_NO := W#16#0;
   S711_WELD_BUFF_DATA71.RBT14_WELD_COUNT := W#16#0;
   S711_WELD_BUFF_DATA71.RBT15_BT_CODE_NO := W#16#0;
   S711_WELD_BUFF_DATA71.RBT15_WELD_COUNT := W#16#0;
   S711_WELD_BUFF_DATA71.RBT16_BT_CODE_NO := W#16#0;
   S711_WELD_BUFF_DATA71.RBT16_WELD_COUNT := W#16#0;
   S711_WELD_BUFF_DATA71.RBT17_BT_CODE_NO := W#16#0;
   S711_WELD_BUFF_DATA71.RBT17_WELD_COUNT := W#16#0;
   S711_WELD_BUFF_DATA71.RBT18_BT_CODE_NO := W#16#0;
   S711_WELD_BUFF_DATA71.RBT18_WELD_COUNT := W#16#0;
   S711_WELD_BUFF_DATA71.RBT19_BT_CODE_NO := W#16#0;
   S711_WELD_BUFF_DATA71.RBT19_WELD_COUNT := W#16#0;
   S711_WELD_BUFF_DATA71.RBT20_BT_CODE_NO := W#16#0;
   S711_WELD_BUFF_DATA71.RBT20_WELD_COUNT := W#16#0;
   S711_WELD_BUFF_DATA71.RBT21_BT_CODE_NO := W#16#0;
   S711_WELD_BUFF_DATA71.RBT21_WELD_COUNT := W#16#0;
   S711_WELD_BUFF_DATA71.RBT22_BT_CODE_NO := W#16#0;
   S711_WELD_BUFF_DATA71.RBT22_WELD_COUNT := W#16#0;
   S711_WELD_BUFF_DATA71.RBT23_BT_CODE_NO := W#16#0;
   S711_WELD_BUFF_DATA71.RBT23_WELD_COUNT := W#16#0;
   S711_WELD_BUFF_DATA71.RBT24_BT_CODE_NO := W#16#0;
   S711_WELD_BUFF_DATA71.RBT24_WELD_COUNT := W#16#0;
   S711_WELD_BUFF_DATA71.WELD_DETERMINES_RESULT := W#16#0;
   S711_WELD_BUFF_DATA71.WELD_CHECK_SUM := W#16#0;
   S711_WELD_BUFF_DATA71.SPARE1 := W#16#0;
   S711_WELD_BUFF_DATA81.STATION_MAIN := W#16#0;
   S711_WELD_BUFF_DATA81.DISTINCTION_LH_RH := W#16#0;
   S711_WELD_BUFF_DATA81.STAION_NUMBER := W#16#0;
   S711_WELD_BUFF_DATA81.VIN_NUMBER1 := W#16#0;
   S711_WELD_BUFF_DATA81.VIN_NUMBER2 := W#16#0;
   S711_WELD_BUFF_DATA81.VIN_NUMBER3 := W#16#0;
   S711_WELD_BUFF_DATA81.VIN_NUMBER4 := W#16#0;
   S711_WELD_BUFF_DATA81.SEQ_NUMBER1 := W#16#0;
   S711_WELD_BUFF_DATA81.SEQ_NUMBER2 := W#16#0;
   S711_WELD_BUFF_DATA81.RBT1_BT_CODE_NO := W#16#0;
   S711_WELD_BUFF_DATA81.RBT1_WELD_COUNT := W#16#0;
   S711_WELD_BUFF_DATA81.RBT2_BT_CODE_NO := W#16#0;
   S711_WELD_BUFF_DATA81.RBT2_WELD_COUNT := W#16#0;
   S711_WELD_BUFF_DATA81.RBT3_BT_CODE_NO := W#16#0;
   S711_WELD_BUFF_DATA81.RBT3_WELD_COUNT := W#16#0;
   S711_WELD_BUFF_DATA81.RBT4_BT_CODE_NO := W#16#0;
   S711_WELD_BUFF_DATA81.RBT4_WELD_COUNT := W#16#0;
   S711_WELD_BUFF_DATA81.RBT5_BT_CODE_NO := W#16#0;
   S711_WELD_BUFF_DATA81.RBT5_WELD_COUNT := W#16#0;
   S711_WELD_BUFF_DATA81.RBT6_BT_CODE_NO := W#16#0;
   S711_WELD_BUFF_DATA81.RBT6_WELD_COUNT := W#16#0;
   S711_WELD_BUFF_DATA81.RBT7_BT_CODE_NO := W#16#0;
   S711_WELD_BUFF_DATA81.RBT7_WELD_COUNT := W#16#0;
   S711_WELD_BUFF_DATA81.RBT8_BT_CODE_NO := W#16#0;
   S711_WELD_BUFF_DATA81.RBT8_WELD_COUNT := W#16#0;
   S711_WELD_BUFF_DATA81.RBT9_BT_CODE_NO := W#16#0;
   S711_WELD_BUFF_DATA81.RBT9_WELD_COUNT := W#16#0;
   S711_WELD_BUFF_DATA81.RBT10_BT_CODE_NO := W#16#0;
   S711_WELD_BUFF_DATA81.RBT10_WELD_COUNT := W#16#0;
   S711_WELD_BUFF_DATA81.RBT11_BT_CODE_NO := W#16#0;
   S711_WELD_BUFF_DATA81.RBT11_WELD_COUNT := W#16#0;
   S711_WELD_BUFF_DATA81.RBT12_BT_CODE_NO := W#16#0;
   S711_WELD_BUFF_DATA81.RBT12_WELD_COUNT := W#16#0;
   S711_WELD_BUFF_DATA81.RBT13_BT_CODE_NO := W#16#0;
   S711_WELD_BUFF_DATA81.RBT13_WELD_COUNT := W#16#0;
   S711_WELD_BUFF_DATA81.RBT14_BT_CODE_NO := W#16#0;
   S711_WELD_BUFF_DATA81.RBT14_WELD_COUNT := W#16#0;
   S711_WELD_BUFF_DATA81.RBT15_BT_CODE_NO := W#16#0;
   S711_WELD_BUFF_DATA81.RBT15_WELD_COUNT := W#16#0;
   S711_WELD_BUFF_DATA81.RBT16_BT_CODE_NO := W#16#0;
   S711_WELD_BUFF_DATA81.RBT16_WELD_COUNT := W#16#0;
   S711_WELD_BUFF_DATA81.RBT17_BT_CODE_NO := W#16#0;
   S711_WELD_BUFF_DATA81.RBT17_WELD_COUNT := W#16#0;
   S711_WELD_BUFF_DATA81.RBT18_BT_CODE_NO := W#16#0;
   S711_WELD_BUFF_DATA81.RBT18_WELD_COUNT := W#16#0;
   S711_WELD_BUFF_DATA81.RBT19_BT_CODE_NO := W#16#0;
   S711_WELD_BUFF_DATA81.RBT19_WELD_COUNT := W#16#0;
   S711_WELD_BUFF_DATA81.RBT20_BT_CODE_NO := W#16#0;
   S711_WELD_BUFF_DATA81.RBT20_WELD_COUNT := W#16#0;
   S711_WELD_BUFF_DATA81.RBT21_BT_CODE_NO := W#16#0;
   S711_WELD_BUFF_DATA81.RBT21_WELD_COUNT := W#16#0;
   S711_WELD_BUFF_DATA81.RBT22_BT_CODE_NO := W#16#0;
   S711_WELD_BUFF_DATA81.RBT22_WELD_COUNT := W#16#0;
   S711_WELD_BUFF_DATA81.RBT23_BT_CODE_NO := W#16#0;
   S711_WELD_BUFF_DATA81.RBT23_WELD_COUNT := W#16#0;
   S711_WELD_BUFF_DATA81.RBT24_BT_CODE_NO := W#16#0;
   S711_WELD_BUFF_DATA81.RBT24_WELD_COUNT := W#16#0;
   S711_WELD_BUFF_DATA81.WELD_DETERMINES_RESULT := W#16#0;
   S711_WELD_BUFF_DATA81.WELD_CHECK_SUM := W#16#0;
   S711_WELD_BUFF_DATA81.SPARE1 := W#16#0;
   S711_WELD_BUFF_DATA91.STATION_MAIN := W#16#0;
   S711_WELD_BUFF_DATA91.DISTINCTION_LH_RH := W#16#0;
   S711_WELD_BUFF_DATA91.STAION_NUMBER := W#16#0;
   S711_WELD_BUFF_DATA91.VIN_NUMBER1 := W#16#0;
   S711_WELD_BUFF_DATA91.VIN_NUMBER2 := W#16#0;
   S711_WELD_BUFF_DATA91.VIN_NUMBER3 := W#16#0;
   S711_WELD_BUFF_DATA91.VIN_NUMBER4 := W#16#0;
   S711_WELD_BUFF_DATA91.SEQ_NUMBER1 := W#16#0;
   S711_WELD_BUFF_DATA91.SEQ_NUMBER2 := W#16#0;
   S711_WELD_BUFF_DATA91.RBT1_BT_CODE_NO := W#16#0;
   S711_WELD_BUFF_DATA91.RBT1_WELD_COUNT := W#16#0;
   S711_WELD_BUFF_DATA91.RBT2_BT_CODE_NO := W#16#0;
   S711_WELD_BUFF_DATA91.RBT2_WELD_COUNT := W#16#0;
   S711_WELD_BUFF_DATA91.RBT3_BT_CODE_NO := W#16#0;
   S711_WELD_BUFF_DATA91.RBT3_WELD_COUNT := W#16#0;
   S711_WELD_BUFF_DATA91.RBT4_BT_CODE_NO := W#16#0;
   S711_WELD_BUFF_DATA91.RBT4_WELD_COUNT := W#16#0;
   S711_WELD_BUFF_DATA91.RBT5_BT_CODE_NO := W#16#0;
   S711_WELD_BUFF_DATA91.RBT5_WELD_COUNT := W#16#0;
   S711_WELD_BUFF_DATA91.RBT6_BT_CODE_NO := W#16#0;
   S711_WELD_BUFF_DATA91.RBT6_WELD_COUNT := W#16#0;
   S711_WELD_BUFF_DATA91.RBT7_BT_CODE_NO := W#16#0;
   S711_WELD_BUFF_DATA91.RBT7_WELD_COUNT := W#16#0;
   S711_WELD_BUFF_DATA91.RBT8_BT_CODE_NO := W#16#0;
   S711_WELD_BUFF_DATA91.RBT8_WELD_COUNT := W#16#0;
   S711_WELD_BUFF_DATA91.RBT9_BT_CODE_NO := W#16#0;
   S711_WELD_BUFF_DATA91.RBT9_WELD_COUNT := W#16#0;
   S711_WELD_BUFF_DATA91.RBT10_BT_CODE_NO := W#16#0;
   S711_WELD_BUFF_DATA91.RBT10_WELD_COUNT := W#16#0;
   S711_WELD_BUFF_DATA91.RBT11_BT_CODE_NO := W#16#0;
   S711_WELD_BUFF_DATA91.RBT11_WELD_COUNT := W#16#0;
   S711_WELD_BUFF_DATA91.RBT12_BT_CODE_NO := W#16#0;
   S711_WELD_BUFF_DATA91.RBT12_WELD_COUNT := W#16#0;
   S711_WELD_BUFF_DATA91.RBT13_BT_CODE_NO := W#16#0;
   S711_WELD_BUFF_DATA91.RBT13_WELD_COUNT := W#16#0;
   S711_WELD_BUFF_DATA91.RBT14_BT_CODE_NO := W#16#0;
   S711_WELD_BUFF_DATA91.RBT14_WELD_COUNT := W#16#0;
   S711_WELD_BUFF_DATA91.RBT15_BT_CODE_NO := W#16#0;
   S711_WELD_BUFF_DATA91.RBT15_WELD_COUNT := W#16#0;
   S711_WELD_BUFF_DATA91.RBT16_BT_CODE_NO := W#16#0;
   S711_WELD_BUFF_DATA91.RBT16_WELD_COUNT := W#16#0;
   S711_WELD_BUFF_DATA91.RBT17_BT_CODE_NO := W#16#0;
   S711_WELD_BUFF_DATA91.RBT17_WELD_COUNT := W#16#0;
   S711_WELD_BUFF_DATA91.RBT18_BT_CODE_NO := W#16#0;
   S711_WELD_BUFF_DATA91.RBT18_WELD_COUNT := W#16#0;
   S711_WELD_BUFF_DATA91.RBT19_BT_CODE_NO := W#16#0;
   S711_WELD_BUFF_DATA91.RBT19_WELD_COUNT := W#16#0;
   S711_WELD_BUFF_DATA91.RBT20_BT_CODE_NO := W#16#0;
   S711_WELD_BUFF_DATA91.RBT20_WELD_COUNT := W#16#0;
   S711_WELD_BUFF_DATA91.RBT21_BT_CODE_NO := W#16#0;
   S711_WELD_BUFF_DATA91.RBT21_WELD_COUNT := W#16#0;
   S711_WELD_BUFF_DATA91.RBT22_BT_CODE_NO := W#16#0;
   S711_WELD_BUFF_DATA91.RBT22_WELD_COUNT := W#16#0;
   S711_WELD_BUFF_DATA91.RBT23_BT_CODE_NO := W#16#0;
   S711_WELD_BUFF_DATA91.RBT23_WELD_COUNT := W#16#0;
   S711_WELD_BUFF_DATA91.RBT24_BT_CODE_NO := W#16#0;
   S711_WELD_BUFF_DATA91.RBT24_WELD_COUNT := W#16#0;
   S711_WELD_BUFF_DATA91.WELD_DETERMINES_RESULT := W#16#0;
   S711_WELD_BUFF_DATA91.WELD_CHECK_SUM := W#16#0;
   S711_WELD_BUFF_DATA91.SPARE1 := W#16#0;
   S711_WELD_BUFF_DATA101.STATION_MAIN := W#16#0;
   S711_WELD_BUFF_DATA101.DISTINCTION_LH_RH := W#16#0;
   S711_WELD_BUFF_DATA101.STAION_NUMBER := W#16#0;
   S711_WELD_BUFF_DATA101.VIN_NUMBER1 := W#16#0;
   S711_WELD_BUFF_DATA101.VIN_NUMBER2 := W#16#0;
   S711_WELD_BUFF_DATA101.VIN_NUMBER3 := W#16#0;
   S711_WELD_BUFF_DATA101.VIN_NUMBER4 := W#16#0;
   S711_WELD_BUFF_DATA101.SEQ_NUMBER1 := W#16#0;
   S711_WELD_BUFF_DATA101.SEQ_NUMBER2 := W#16#0;
   S711_WELD_BUFF_DATA101.RBT1_BT_CODE_NO := W#16#0;
   S711_WELD_BUFF_DATA101.RBT1_WELD_COUNT := W#16#0;
   S711_WELD_BUFF_DATA101.RBT2_BT_CODE_NO := W#16#0;
   S711_WELD_BUFF_DATA101.RBT2_WELD_COUNT := W#16#0;
   S711_WELD_BUFF_DATA101.RBT3_BT_CODE_NO := W#16#0;
   S711_WELD_BUFF_DATA101.RBT3_WELD_COUNT := W#16#0;
   S711_WELD_BUFF_DATA101.RBT4_BT_CODE_NO := W#16#0;
   S711_WELD_BUFF_DATA101.RBT4_WELD_COUNT := W#16#0;
   S711_WELD_BUFF_DATA101.RBT5_BT_CODE_NO := W#16#0;
   S711_WELD_BUFF_DATA101.RBT5_WELD_COUNT := W#16#0;
   S711_WELD_BUFF_DATA101.RBT6_BT_CODE_NO := W#16#0;
   S711_WELD_BUFF_DATA101.RBT6_WELD_COUNT := W#16#0;
   S711_WELD_BUFF_DATA101.RBT7_BT_CODE_NO := W#16#0;
   S711_WELD_BUFF_DATA101.RBT7_WELD_COUNT := W#16#0;
   S711_WELD_BUFF_DATA101.RBT8_BT_CODE_NO := W#16#0;
   S711_WELD_BUFF_DATA101.RBT8_WELD_COUNT := W#16#0;
   S711_WELD_BUFF_DATA101.RBT9_BT_CODE_NO := W#16#0;
   S711_WELD_BUFF_DATA101.RBT9_WELD_COUNT := W#16#0;
   S711_WELD_BUFF_DATA101.RBT10_BT_CODE_NO := W#16#0;
   S711_WELD_BUFF_DATA101.RBT10_WELD_COUNT := W#16#0;
   S711_WELD_BUFF_DATA101.RBT11_BT_CODE_NO := W#16#0;
   S711_WELD_BUFF_DATA101.RBT11_WELD_COUNT := W#16#0;
   S711_WELD_BUFF_DATA101.RBT12_BT_CODE_NO := W#16#0;
   S711_WELD_BUFF_DATA101.RBT12_WELD_COUNT := W#16#0;
   S711_WELD_BUFF_DATA101.RBT13_BT_CODE_NO := W#16#0;
   S711_WELD_BUFF_DATA101.RBT13_WELD_COUNT := W#16#0;
   S711_WELD_BUFF_DATA101.RBT14_BT_CODE_NO := W#16#0;
   S711_WELD_BUFF_DATA101.RBT14_WELD_COUNT := W#16#0;
   S711_WELD_BUFF_DATA101.RBT15_BT_CODE_NO := W#16#0;
   S711_WELD_BUFF_DATA101.RBT15_WELD_COUNT := W#16#0;
   S711_WELD_BUFF_DATA101.RBT16_BT_CODE_NO := W#16#0;
   S711_WELD_BUFF_DATA101.RBT16_WELD_COUNT := W#16#0;
   S711_WELD_BUFF_DATA101.RBT17_BT_CODE_NO := W#16#0;
   S711_WELD_BUFF_DATA101.RBT17_WELD_COUNT := W#16#0;
   S711_WELD_BUFF_DATA101.RBT18_BT_CODE_NO := W#16#0;
   S711_WELD_BUFF_DATA101.RBT18_WELD_COUNT := W#16#0;
   S711_WELD_BUFF_DATA101.RBT19_BT_CODE_NO := W#16#0;
   S711_WELD_BUFF_DATA101.RBT19_WELD_COUNT := W#16#0;
   S711_WELD_BUFF_DATA101.RBT20_BT_CODE_NO := W#16#0;
   S711_WELD_BUFF_DATA101.RBT20_WELD_COUNT := W#16#0;
   S711_WELD_BUFF_DATA101.RBT21_BT_CODE_NO := W#16#0;
   S711_WELD_BUFF_DATA101.RBT21_WELD_COUNT := W#16#0;
   S711_WELD_BUFF_DATA101.RBT22_BT_CODE_NO := W#16#0;
   S711_WELD_BUFF_DATA101.RBT22_WELD_COUNT := W#16#0;
   S711_WELD_BUFF_DATA101.RBT23_BT_CODE_NO := W#16#0;
   S711_WELD_BUFF_DATA101.RBT23_WELD_COUNT := W#16#0;
   S711_WELD_BUFF_DATA101.RBT24_BT_CODE_NO := W#16#0;
   S711_WELD_BUFF_DATA101.RBT24_WELD_COUNT := W#16#0;
   S711_WELD_BUFF_DATA101.WELD_DETERMINES_RESULT := W#16#0;
   S711_WELD_BUFF_DATA101.WELD_CHECK_SUM := W#16#0;
   S711_WELD_BUFF_DATA101.SPARE1 := W#16#0;
END_DATA_BLOCK

DATA_BLOCK DB 45
TITLE =
VERSION : 0.1


  STRUCT
   STAT0 : ARRAY  [0 .. 300 ] OF WORD  := W#16#0;
  END_STRUCT ;
BEGIN
   STAT0[0] := W#16#0;
   STAT0[1] := W#16#0;
   STAT0[2] := W#16#0;
   STAT0[3] := W#16#0;
   STAT0[4] := W#16#0;
   STAT0[5] := W#16#0;
   STAT0[6] := W#16#0;
   STAT0[7] := W#16#0;
   STAT0[8] := W#16#0;
   STAT0[9] := W#16#0;
   STAT0[10] := W#16#0;
   STAT0[11] := W#16#0;
   STAT0[12] := W#16#0;
   STAT0[13] := W#16#0;
   STAT0[14] := W#16#0;
   STAT0[15] := W#16#0;
   STAT0[16] := W#16#0;
   STAT0[17] := W#16#0;
   STAT0[18] := W#16#0;
   STAT0[19] := W#16#0;
   STAT0[20] := W#16#0;
   STAT0[21] := W#16#0;
   STAT0[22] := W#16#0;
   STAT0[23] := W#16#0;
   STAT0[24] := W#16#0;
   STAT0[25] := W#16#0;
   STAT0[26] := W#16#0;
   STAT0[27] := W#16#0;
   STAT0[28] := W#16#0;
   STAT0[29] := W#16#0;
   STAT0[30] := W#16#0;
   STAT0[31] := W#16#0;
   STAT0[32] := W#16#0;
   STAT0[33] := W#16#0;
   STAT0[34] := W#16#0;
   STAT0[35] := W#16#0;
   STAT0[36] := W#16#0;
   STAT0[37] := W#16#0;
   STAT0[38] := W#16#0;
   STAT0[39] := W#16#0;
   STAT0[40] := W#16#0;
   STAT0[41] := W#16#0;
   STAT0[42] := W#16#0;
   STAT0[43] := W#16#0;
   STAT0[44] := W#16#0;
   STAT0[45] := W#16#0;
   STAT0[46] := W#16#0;
   STAT0[47] := W#16#0;
   STAT0[48] := W#16#0;
   STAT0[49] := W#16#0;
   STAT0[50] := W#16#0;
   STAT0[51] := W#16#0;
   STAT0[52] := W#16#0;
   STAT0[53] := W#16#0;
   STAT0[54] := W#16#0;
   STAT0[55] := W#16#0;
   STAT0[56] := W#16#0;
   STAT0[57] := W#16#0;
   STAT0[58] := W#16#0;
   STAT0[59] := W#16#0;
   STAT0[60] := W#16#0;
   STAT0[61] := W#16#0;
   STAT0[62] := W#16#0;
   STAT0[63] := W#16#0;
   STAT0[64] := W#16#0;
   STAT0[65] := W#16#0;
   STAT0[66] := W#16#0;
   STAT0[67] := W#16#0;
   STAT0[68] := W#16#0;
   STAT0[69] := W#16#0;
   STAT0[70] := W#16#0;
   STAT0[71] := W#16#0;
   STAT0[72] := W#16#0;
   STAT0[73] := W#16#0;
   STAT0[74] := W#16#0;
   STAT0[75] := W#16#0;
   STAT0[76] := W#16#0;
   STAT0[77] := W#16#0;
   STAT0[78] := W#16#0;
   STAT0[79] := W#16#0;
   STAT0[80] := W#16#0;
   STAT0[81] := W#16#0;
   STAT0[82] := W#16#0;
   STAT0[83] := W#16#0;
   STAT0[84] := W#16#0;
   STAT0[85] := W#16#0;
   STAT0[86] := W#16#0;
   STAT0[87] := W#16#0;
   STAT0[88] := W#16#0;
   STAT0[89] := W#16#0;
   STAT0[90] := W#16#0;
   STAT0[91] := W#16#0;
   STAT0[92] := W#16#0;
   STAT0[93] := W#16#0;
   STAT0[94] := W#16#0;
   STAT0[95] := W#16#0;
   STAT0[96] := W#16#0;
   STAT0[97] := W#16#0;
   STAT0[98] := W#16#0;
   STAT0[99] := W#16#0;
   STAT0[100] := W#16#0;
   STAT0[101] := W#16#0;
   STAT0[102] := W#16#0;
   STAT0[103] := W#16#0;
   STAT0[104] := W#16#0;
   STAT0[105] := W#16#0;
   STAT0[106] := W#16#0;
   STAT0[107] := W#16#0;
   STAT0[108] := W#16#0;
   STAT0[109] := W#16#0;
   STAT0[110] := W#16#0;
   STAT0[111] := W#16#0;
   STAT0[112] := W#16#0;
   STAT0[113] := W#16#0;
   STAT0[114] := W#16#0;
   STAT0[115] := W#16#0;
   STAT0[116] := W#16#0;
   STAT0[117] := W#16#0;
   STAT0[118] := W#16#0;
   STAT0[119] := W#16#0;
   STAT0[120] := W#16#0;
   STAT0[121] := W#16#0;
   STAT0[122] := W#16#0;
   STAT0[123] := W#16#0;
   STAT0[124] := W#16#0;
   STAT0[125] := W#16#0;
   STAT0[126] := W#16#0;
   STAT0[127] := W#16#0;
   STAT0[128] := W#16#0;
   STAT0[129] := W#16#0;
   STAT0[130] := W#16#0;
   STAT0[131] := W#16#0;
   STAT0[132] := W#16#0;
   STAT0[133] := W#16#0;
   STAT0[134] := W#16#0;
   STAT0[135] := W#16#0;
   STAT0[136] := W#16#0;
   STAT0[137] := W#16#0;
   STAT0[138] := W#16#0;
   STAT0[139] := W#16#0;
   STAT0[140] := W#16#0;
   STAT0[141] := W#16#0;
   STAT0[142] := W#16#0;
   STAT0[143] := W#16#0;
   STAT0[144] := W#16#0;
   STAT0[145] := W#16#0;
   STAT0[146] := W#16#0;
   STAT0[147] := W#16#0;
   STAT0[148] := W#16#0;
   STAT0[149] := W#16#0;
   STAT0[150] := W#16#0;
   STAT0[151] := W#16#0;
   STAT0[152] := W#16#0;
   STAT0[153] := W#16#0;
   STAT0[154] := W#16#0;
   STAT0[155] := W#16#0;
   STAT0[156] := W#16#0;
   STAT0[157] := W#16#0;
   STAT0[158] := W#16#0;
   STAT0[159] := W#16#0;
   STAT0[160] := W#16#0;
   STAT0[161] := W#16#0;
   STAT0[162] := W#16#0;
   STAT0[163] := W#16#0;
   STAT0[164] := W#16#0;
   STAT0[165] := W#16#0;
   STAT0[166] := W#16#0;
   STAT0[167] := W#16#0;
   STAT0[168] := W#16#0;
   STAT0[169] := W#16#0;
   STAT0[170] := W#16#0;
   STAT0[171] := W#16#0;
   STAT0[172] := W#16#0;
   STAT0[173] := W#16#0;
   STAT0[174] := W#16#0;
   STAT0[175] := W#16#0;
   STAT0[176] := W#16#0;
   STAT0[177] := W#16#0;
   STAT0[178] := W#16#0;
   STAT0[179] := W#16#0;
   STAT0[180] := W#16#0;
   STAT0[181] := W#16#0;
   STAT0[182] := W#16#0;
   STAT0[183] := W#16#0;
   STAT0[184] := W#16#0;
   STAT0[185] := W#16#0;
   STAT0[186] := W#16#0;
   STAT0[187] := W#16#0;
   STAT0[188] := W#16#0;
   STAT0[189] := W#16#0;
   STAT0[190] := W#16#0;
   STAT0[191] := W#16#0;
   STAT0[192] := W#16#0;
   STAT0[193] := W#16#0;
   STAT0[194] := W#16#0;
   STAT0[195] := W#16#0;
   STAT0[196] := W#16#0;
   STAT0[197] := W#16#0;
   STAT0[198] := W#16#0;
   STAT0[199] := W#16#0;
   STAT0[200] := W#16#0;
   STAT0[201] := W#16#0;
   STAT0[202] := W#16#0;
   STAT0[203] := W#16#0;
   STAT0[204] := W#16#0;
   STAT0[205] := W#16#0;
   STAT0[206] := W#16#0;
   STAT0[207] := W#16#0;
   STAT0[208] := W#16#0;
   STAT0[209] := W#16#0;
   STAT0[210] := W#16#0;
   STAT0[211] := W#16#0;
   STAT0[212] := W#16#0;
   STAT0[213] := W#16#0;
   STAT0[214] := W#16#0;
   STAT0[215] := W#16#0;
   STAT0[216] := W#16#0;
   STAT0[217] := W#16#0;
   STAT0[218] := W#16#0;
   STAT0[219] := W#16#0;
   STAT0[220] := W#16#0;
   STAT0[221] := W#16#0;
   STAT0[222] := W#16#0;
   STAT0[223] := W#16#0;
   STAT0[224] := W#16#0;
   STAT0[225] := W#16#0;
   STAT0[226] := W#16#0;
   STAT0[227] := W#16#0;
   STAT0[228] := W#16#0;
   STAT0[229] := W#16#0;
   STAT0[230] := W#16#0;
   STAT0[231] := W#16#0;
   STAT0[232] := W#16#0;
   STAT0[233] := W#16#0;
   STAT0[234] := W#16#0;
   STAT0[235] := W#16#0;
   STAT0[236] := W#16#0;
   STAT0[237] := W#16#0;
   STAT0[238] := W#16#0;
   STAT0[239] := W#16#0;
   STAT0[240] := W#16#0;
   STAT0[241] := W#16#0;
   STAT0[242] := W#16#0;
   STAT0[243] := W#16#0;
   STAT0[244] := W#16#0;
   STAT0[245] := W#16#0;
   STAT0[246] := W#16#0;
   STAT0[247] := W#16#0;
   STAT0[248] := W#16#0;
   STAT0[249] := W#16#0;
   STAT0[250] := W#16#0;
   STAT0[251] := W#16#0;
   STAT0[252] := W#16#0;
   STAT0[253] := W#16#0;
   STAT0[254] := W#16#0;
   STAT0[255] := W#16#0;
   STAT0[256] := W#16#0;
   STAT0[257] := W#16#0;
   STAT0[258] := W#16#0;
   STAT0[259] := W#16#0;
   STAT0[260] := W#16#0;
   STAT0[261] := W#16#0;
   STAT0[262] := W#16#0;
   STAT0[263] := W#16#0;
   STAT0[264] := W#16#0;
   STAT0[265] := W#16#0;
   STAT0[266] := W#16#0;
   STAT0[267] := W#16#0;
   STAT0[268] := W#16#0;
   STAT0[269] := W#16#0;
   STAT0[270] := W#16#0;
   STAT0[271] := W#16#0;
   STAT0[272] := W#16#0;
   STAT0[273] := W#16#0;
   STAT0[274] := W#16#0;
   STAT0[275] := W#16#0;
   STAT0[276] := W#16#0;
   STAT0[277] := W#16#0;
   STAT0[278] := W#16#0;
   STAT0[279] := W#16#0;
   STAT0[280] := W#16#0;
   STAT0[281] := W#16#0;
   STAT0[282] := W#16#0;
   STAT0[283] := W#16#0;
   STAT0[284] := W#16#0;
   STAT0[285] := W#16#0;
   STAT0[286] := W#16#0;
   STAT0[287] := W#16#0;
   STAT0[288] := W#16#0;
   STAT0[289] := W#16#0;
   STAT0[290] := W#16#0;
   STAT0[291] := W#16#0;
   STAT0[292] := W#16#0;
   STAT0[293] := W#16#0;
   STAT0[294] := W#16#0;
   STAT0[295] := W#16#0;
   STAT0[296] := W#16#0;
   STAT0[297] := W#16#0;
   STAT0[298] := W#16#0;
   STAT0[299] := W#16#0;
   STAT0[300] := W#16#0;
END_DATA_BLOCK

DATA_BLOCK DB 51
TITLE =
VERSION : 0.1


